		IF stOuterStatus.stOACData.PackCodeStatus[nPackIndex].5 OR stOuterStatus.stOACData.PackCodeStatus[nPackIndex].6 THEN

			FOR nCheckIndex :=1 TO cMAX_PACKS_PER_OUTER DO

				IF stOuterStatus.stOACData.PackCode[nPackIndex] = stLastOuterStatus.stOACData.PackCode[nCheckIndex] THEN

					stOuterStatus.nStatus.22 := TRUE;
					stOuterStatus.sDataSourceTracker  := 'PK_DUPLIC';

					stLastOuterStatus.nStatus.22 := TRUE;
					stLastOuterStatus.sDataSourceTracker  := 'PK_DUPLIC';

					EXIT;
				END_IF
			END_FOR
			EXIT;
		END_IF
	END_FOR
END_IF

bDuplicateFound 	:= FALSE;

(* for dupicats for all packs inside one Outer *)
FOR  nPackIndex :=1 TO cMAX_PACKS_PER_OUTER DO

	IF stOuterStatus.stOACData.PackCodeStatus[nPackIndex].5 OR stOuterStatus.stOACData.PackCodeStatus[nPackIndex].6 THEN

		FOR nCheckIndex := nPackIndex  TO cMAX_PACKS_PER_OUTER DO

			IF stOuterStatus.stOACData.PackCodeStatus[nCheckIndex].5 OR stOuterStatus.stOACData.PackCodeStatus[nCheckIndex].6 THEN

				IF stOuterStatus.stOACData.PackCode[nPackIndex] = stOuterStatus.stOACData.PackCode[nCheckIndex]  AND
					nPackIndex <> nCheckIndex	THEN


					(* duplicate packs found *)
					stOuterStatus.aOACPackStatus[nPackIndex] := 3;
					(*additional bit passing to CAC*)
					stOuterStatus.stOACData.PackCodeStatus[nPackIndex] :=
											F_FiltredSetBitState16(TRUE, 'LOW', 3, TRUE, stOuterStatus.stOACData.PackCodeStatus[nPackIndex]);

					stOuterStatus.aOACPackStatus[nCheckIndex] := 3;
					(*additional bit passing to CAC*)
					stOuterStatus.stOACData.PackCodeStatus[nCheckIndex] :=
											F_FiltredSetBitState16(TRUE, 'LOW', 3, TRUE, stOuterStatus.stOACData.PackCodeStatus[nCheckIndex]);

					bDuplicateFound := TRUE;

					stOuterStatus.stOACData.PackRejectCode[nPackIndex]  	:= stDuplicatedItem.sMetsDisplayCode;
	   				stOuterStatus.stOACData.PackRejectID[nPackIndex] 	 	:= stDuplicatedItem.nRejectID;
					stOuterStatus.stOACData.PackRejectCode[nCheckIndex]  := stDuplicatedItem.sMetsDisplayCode;
					stOuterStatus.stOACData.PackRejectID[nCheckIndex]  	:= stDuplicatedItem.nRejectID;

				END_IF
			END_IF
		END_FOR
	END_IF
END_FOR


IF bDuplicateFound THEN

	nGoodPackReads	:=cMAX_PACKS_PER_OUTER;
	stOuterStatus.nStatus.23 := TRUE;

	FOR  nPackIndex :=1 TO cMAX_PACKS_PER_OUTER DO
		IF stOuterStatus.stOACData.PackCodeStatus[nPackIndex].3 THEN nGoodPackReads := nGoodPackReads - 1; END_IF
	END_FOR

END_IF

END_FUNCTION_BLOCK

// ---- POUs/METS/Common LIB/01_PACK LIB/Pack FBs/FB_PACK_MoveOuterStatusArray.TcPOU
FUNCTION_BLOCK FB_PACK_MoveOuterStatusArray
VAR_INPUT
	bExecute			: BOOL;		(* set TRUE to move array data *)
	bClearShiftReg		: BOOL;		(* set TRUE to clear all array data to 0 *)
END_VAR
VAR_IN_OUT
	aOCVPackStatus			: ARRAY[1..cMAX_OUTER_STATUS_QUEUE] OF ST_OUTER_Status;	(* Outer status register *)
	(*stPackBufferStatusHMI		: ST_HMI_PACK_BufferStatus;*)
END_VAR
VAR_OUTPUT
	bDone						: BOOL;
END_VAR
VAR
	fbExecute			: R_TRIG;
END_VAR

(* rising edge of bShiftReg *)
fbExecute(CLK := bExecute);

(* clear shift reg *)
IF bClearShiftReg = TRUE THEN

	(* reset OCV Outer Status data *)
	MEMSET(ADR(aOCVPackStatus), 16#00, SIZEOF(aOCVPackStatus));

	bDone := FALSE;

(* move shift reg *)
ELSIF fbExecute.Q = TRUE THEN

	(* move OCV Outer Status register [1..cMAX_OUTER_STATUS_QUEUE-1] to [2..cMAX_OUTER_STATUS_QUEUE] *)
	MEMMOVE(ADR(aOCVPackStatus[2]), ADR(aOCVPackStatus[1]), SIZEOF(aOCVPackStatus) - SIZEOF(aOCVPackStatus[1]));
	(* clear OCV Outer Status register [1] *)
	MEMSET(ADR(aOCVPackStatus[1]), 16#00, SIZEOF(aOCVPackStatus[1]));

	(*MEMSET(ADR(stPackBufferStatusHMI), 16#00, SIZEOF(stPackBufferStatusHMI));*)

	bDone := TRUE;

(* no action required, bExecute has been reset *)
ELSIF bExecute = FALSE THEN

	bDone := FALSE;
END_IF

(******************************************************************************************************************************************)
(*
IN CASE OF MULTISHIFT - CAN BE USED THIS:
	nOuterStatusToShift := LIMIT(1, nOuterStatusToShift, cMAX_OUTER_STATUS_QUEUE);
	(* move Outer Status register [1..49] to [2..50] *)
	MEMMOVE(ADR(aOuterStatus[nOuterStatusToShift+1]), ADR(aOuterStatus[1]), SIZEOF(aOuterStatus) - nOuterStatusToShift*SIZEOF(aOuterStatus[1]));
	(* clear Outer Status register [nOuterStatusToShift] *)
	MEMSET(ADR(aOuterStatus[1]), 16#00, nOuterStatusToShift*SIZEOF(aOuterStatus[1]));
*)
(******************************************************************************************************************************************)

END_FUNCTION_BLOCK

// ---- POUs/METS/Common LIB/01_PACK LIB/Pack FBs/FB_PACK_WriteOCVLoopDB.TcPOU
(* scan and validate Outers, generate OAC file for new valid Outers *)
FUNCTION_BLOCK FB_PACK_WriteOCVLoopDB
VAR_INPUT
	bExecute						: BOOL;			(* scan for completed Outer *)
	ePackAggregationMode			: E_SYSTEM_PackAggregationMode ;
	nPacksPerOuter				: INT;
	nPackPos1						: INT 	:=1;
	nPackPos2						: INT	:=2;
	bExtendedDupCheck			: BOOL;
	aDisablePackAggregCamera	: ARRAY[1..3] OF BOOL;
	stDuplicatedItem				: ST_RejectItems;(*stPackRejectReasons.stPackCodesDuplicated*)
	stCTDateTime					: ST_SYSTEM_DateTime;
END_VAR
VAR_IN_OUT
	stOCVDataDB					: ST_DB_OCVDataCtrl;
	stLastOCVDataDB				: ST_DB_OCVDataCtrl;
	stCodeInfo_Pack				: ST_CodeInfo;
	stCodeInfo_Intermediate		: ST_CodeInfo;
	(*aInterimCodeQueue			: ARRAY[1..cMAX_INTERMEDIATE_CODE_QUEUE] OF T_MaxString;*)
	aOCVPackStatus				: ARRAY[1..cMAX_OUTER_STATUS_QUEUE] OF ST_OUTER_Status;	(* Outer status array *)
	stMetsEfficiency				: ST_NOVRAM_METS_Inspection;
	stShiftItemProduced			: ST_KPI_ItemsProduced;
	stProdItemProduced			: ST_KPI_ItemsProduced;
	stLastOCVStatus				: ST_OUTER_Status;	(* Outer status *)
END_VAR
VAR_OUTPUT
	bDone							: BOOL;			(* TRUE = validation complete *)
	bBusy							: BOOL;			(* TRUE = validation in progress *)
	bError							: BOOL;			(* TRUE = validation error *)
	nErrorID						: UDINT;			(* error ID *)

	aOCVRecordDBName			 : ARRAY[1..2] OF T_MaxString;

	bPackCodeDuplicate			: BOOL;
	nLastTriggerID					: UDINT;
	bOCVUpdated					: BOOL;
	bOCVValidated					: BOOL;
	stLastValidatedOCV			: ST_OUTER_Status;	(* Outer status *)
	sPackCodesResultToOCV		: T_LongSTRING;
END_VAR
VAR
	fbExecute					: R_TRIG;
	tonTimeOut				: TON;
	rtTimeOutExec				: R_TRIG;
	eState						: E_OCV_State;
	eErrorState					: E_OCV_State;
	eCodeAIType				: E_CodeAIType;
	nMaxOuterIndex			: INT;
	nOuterIndex				: INT;
	nSourceIndex				: INT;
	nPackIndex				: INT;

	nOCVDataCreated 			: UDINT;
	nOCVStoredInDB 			: UDINT;
	nOCVFaildInDB				: UDINT;
	nLinkedPackInOCV 		: UDINT;

	nOCVUpdatedInDB 		: UDINT;

	bUseIntermediateCode		: BOOL;
	stOCVStatus				: ST_OUTER_Status;	(* Outer status *)

(******************************************************************************)

	fbDuplicatesPackCodesDB		: FB_PACK_DuplicatesPackCodesDB;
	fbPackInspectionEfficency		: FB_KPI_PackEfficiency;

(******************************************************************************)

	aDiagOCVDataDB				: ARRAY[0..1] OF ST_DB_OCVDataCtrl;

	nOCVLogIndex		: T_PositiveINT;
	sAppendedString				: STRING;
	//sLocalTargetPath	: T_MaxString;

END_VAR

(***************************************TimeOut *******************************************)
(* monitor Busy timeout *)
tonTimeOut( IN:=nSourceIndex <> 0, PT:=cONE_SECOND, Q=>);

rtTimeOutExec(CLK:= tonTimeOut.Q);

IF rtTimeOutExec.Q THEN

	bError := TRUE;
	nErrorID := 100;
	IF nSourceIndex > 0 THEN

		aOCVPackStatus[nSourceIndex].sDataSourceTracker 	:= 	'TIMEOUT_S';
		aOCVPackStatus[nSourceIndex].nStatus.7 := TRUE;

		stLastOCVStatus := aOCVPackStatus[nSourceIndex];
		bOCVUpdated	:= TRUE;
		sPackCodesResultToOCV	:= 'TIMEOUT_OCV';

		stLastValidatedOCV := aOCVPackStatus[nSourceIndex];
		bOCVValidated	:= TRUE;
	END_IF

	MEMSET(ADR(stOCVDataDB), 16#00, SIZEOF(stOCVDataDB));
	MEMSET(ADR(stLastOCVDataDB), 16#00, SIZEOF(stLastOCVDataDB));


	eState := E_OCV_DONE;
END_IF

(***************************************Execution*******************************************)

(* monitor rising edge of bExecute *)
fbExecute(CLK := bExecute);

(* rising edge of bExecute *)
CASE eState OF

	(* idle *)
	E_OCV_IDLE:

		(* scan for completed Outer when OAC files are required *)
		IF fbExecute.Q = TRUE THEN

			(* update outputs *)
			bDone := FALSE;
			bBusy := TRUE;
			bError := FALSE;
			nErrorID := 0;

			(* clear outputs *)
			nOCVDataCreated 		:= 0;
			nOCVStoredInDB 		:= 0;
			nOCVFaildInDB			:= 0;
			nLinkedPackInOCV 	:= 0;


			(*bOCVUpdated	:= FALSE;*)

			(* max Outer index *)
			nMaxOuterIndex := UDINT_TO_INT(SIZEOF(aOCVPackStatus) / SIZEOF(aOCVPackStatus[1]));

			eState := E_OCV_SCAN;

		(* no action required *)
		ELSIF bExecute = FALSE THEN

			(* reset outputs *)
			bDone := FALSE;
			bBusy := FALSE;
			bError := FALSE;
			nErrorID := 0;

		END_IF

	(* scan for completed Outer *)
	E_OCV_SCAN:

		eState := E_OCV_DONE;
		bOCVUpdated	:= FALSE;
		bOCVValidated	:= FALSE;

		(* reset index of Outer to be written to OCV file *)
		nSourceIndex := 0;

		aOCVRecordDBName[1] := '';
		aOCVRecordDBName[2] := '';

		bPackCodeDuplicate			:= FALSE;

		 (* scan aOCVPackStatus  backward - ensures that oldest Outer will be written first *)
		FOR nOuterIndex := nMaxOuterIndex TO 1 BY -1 DO
			CASE ePackAggregationMode OF

			E_SYSTEM_PAOL_3CAM:
				(* TriggerID > 0 indicates Outer data present, nStatus = 14 indicates writing data for all 3 cameras, nStatus.6  indicates OCV file has been alread  created, nStatus.7 indicates OCV write error  *)
				IF aOCVPackStatus[nOuterIndex].nTriggerID > 0 AND
					(aOCVPackStatus[nOuterIndex].nStatus.1 OR aDisablePackAggregCamera[1])	AND
					( aOCVPackStatus[nOuterIndex].nStatus.2 OR aDisablePackAggregCamera[2]) 	AND
					( aOCVPackStatus[nOuterIndex].nStatus.3 OR aDisablePackAggregCamera[3]) 	AND
					NOT aOCVPackStatus[nOuterIndex].nStatus.6 		AND
					NOT aOCVPackStatus[nOuterIndex].nStatus.7  		(*AND
					NOT aOCVPackStatus[nOuterIndex].nStatus.22		AND
					NOT aOCVPackStatus[nOuterIndex].nStatus.23 *)	THEN

					(* For lightbox system,mapping packcodes to AggregationCodes, used for file name has to be done here, when we are sure if all pack data was plced to OCV record. Those codes will be used to restore OCV data to OAC*)
					AggregationCodes();

					bUseIntermediateCode := FALSE;
					nSourceIndex := nOuterIndex;
					EXIT;
				END_IF

			E_SYSTEM_PAOL_2CAM:
				(* TriggerID > 0 indicates Outer data present, nStatus = 14 indicates writing data for all 3 cameras, nStatus.6  indicates OCV file has been alread  created, nStatus.7 indicates OCV write error  *)
				IF aOCVPackStatus[nOuterIndex].nTriggerID > 0 AND
					(aOCVPackStatus[nOuterIndex].nStatus.1 OR aDisablePackAggregCamera[1])		AND
					( aOCVPackStatus[nOuterIndex].nStatus.2 OR aDisablePackAggregCamera[2]) 	AND
					NOT aOCVPackStatus[nOuterIndex].nStatus.6 		AND
					NOT aOCVPackStatus[nOuterIndex].nStatus.7  		(*AND
					NOT aOCVPackStatus[nOuterIndex].nStatus.22		AND
					NOT aOCVPackStatus[nOuterIndex].nStatus.23*) 	THEN

					(* For lightbox system,mapping packcodes to AggregationCodes, used for file name has to be done here, when we are sure if all pack data was plced to OCV record. Those codes will be used to restore OCV data to OAC*)
					AggregationCodes();

					bUseIntermediateCode := FALSE;
					nSourceIndex := nOuterIndex;
					EXIT;
				END_IF

			E_SYSTEM_PLAS_T01:
				(* TriggerID > 0 indicates Outer data present, nStatus = 14 indicates writing data for all 3 cameras, nStatus.6  indicates OCV file has been alread  created, nStatus.7 indicates OCV write error  *)
				(* For linear aggregation system,AggregationCode shuld be already add from temporary coding system camera. This code will be used for file name and to restore OCV data to OAC*)

				IF aOCVPackStatus[nOuterIndex].nTriggerID > 0 		AND
					aOCVPackStatus[nOuterIndex].nStatus.0			AND 	(*OCV Structure rady to store in file *)
					NOT aOCVPackStatus[nOuterIndex].nStatus.6 		AND
					NOT aOCVPackStatus[nOuterIndex].nStatus.7  		(*AND
					NOT aOCVPackStatus[nOuterIndex].nStatus.22		AND
					NOT aOCVPackStatus[nOuterIndex].nStatus.23 *)	THEN

					(* For clear wrap system,mapping packcodes to AggregationCodes, used for file name has to be done here, when we are sure if all pack data was plced to OCV record. Those codes will be used to restore OCV data to OAC*)
					AggregationCodes();

					bUseIntermediateCode := FALSE;
					nSourceIndex := nOuterIndex;
					EXIT;
				END_IF

			E_SYSTEM_PLAS_T02, E_SYSTEM_PLAS_T03, E_SYSTEM_PLAS_T04:
				(* TriggerID > 0 indicates Outer data present, nStatus = 14 indicates writing data for all 3 cameras, nStatus.6  indicates OCV file has been alread  created, nStatus.7 indicates OCV write error  *)
				(* For linear aggregation system,AggregationCode shuld be already add from temporary coding system camera. This code will be used for file name and to restore OCV data to OAC*)

				IF aOCVPackStatus[nOuterIndex].nTriggerID > 0 		AND
					aOCVPackStatus[nOuterIndex].nStatus.0			AND 	(*OCV Structure rady to store in file *)
					NOT aOCVPackStatus[nOuterIndex].nStatus.6 		AND
					NOT aOCVPackStatus[nOuterIndex].nStatus.7  		(*AND
					NOT aOCVPackStatus[nOuterIndex].nStatus.22		AND
					NOT aOCVPackStatus[nOuterIndex].nStatus.23 *)	THEN

					(* For NON clear wrap system,mapping packcodes to AggregationCodes form Intrim code, which might be temp stored as barcode for OCV records.
						AggregationCode1 will be used for file name has to be done here, when we are sure if all pack data was plced to OCV record. Those codes will be used to restore OCV data to OAC*)
						(*aOCVPackStatus[nOuterIndex].stOACData.AggregationCodes[1] :=aOCVPackStatus[nOuterIndex].stOACData.Barcode;*) (*solution never tested yet*)

					bUseIntermediateCode := TRUE;
					nSourceIndex := nOuterIndex;
					EXIT;
				END_IF
			END_CASE
		END_FOR

		(* Outer found requiring OAC file to be written *)
		IF nSourceIndex > 0 THEN

			(* copy Outer data from arrOuterStatus *)
			stOCVStatus := aOCVPackStatus[nSourceIndex];

			fbDuplicatesPackCodesDB(
				stDuplicatedItem := stDuplicatedItem,
				bExtendedDupCheck	:=	bExtendedDupCheck,
				stOuterStatus := stOCVStatus,
				stLastOuterStatus := aOCVPackStatus[nSourceIndex+1],
				bDuplicateFound =>  bPackCodeDuplicate
				);

			stMetsEfficiency.OutersProcessing.AtPackAggregCameras := stMetsEfficiency.OutersProcessing.AtPackAggregCameras  + 1;

			fbPackInspectionEfficency(
				ePackAggregationMode				:= ePackAggregationMode,
				nTotalOutersProcessingByPackAggregCameras	:= stMetsEfficiency.OutersProcessing.AtPackAggregCameras,
				bUseInterimCode						:= bUseIntermediateCode,
				sOuterStatus							:= stOCVStatus,
				aPacksRead							:= stMetsEfficiency.PacksRead,
				aPackPosEfficiency						:= stMetsEfficiency.PackPosEfficiency,
				stPackAggregationEfficiency			:= stMetsEfficiency.PackAggregationEfficiency,
				stMainItemProduced					:= stMetsEfficiency.PackProduced,
				stShiftItemProduced					:= stShiftItemProduced,
				stProdItemProduced					:= stProdItemProduced
				);

			nOCVDataCreated := nOCVDataCreated +1;

			stLastValidatedOCV := stOCVStatus; (*Use for logging data*)
			bOCVValidated	:= TRUE;	(*Use for SFLX solution*)

			IF aOCVPackStatus[nSourceIndex+1].nStatus.22 AND stOCVStatus.nStatus.22  AND nSourceIndex <  nMaxOuterIndex  THEN

				stLastOCVDataDB.stOCVStatusDB	:= aOCVPackStatus[nSourceIndex+1];
				stLastOCVDataDB.bBlockRecord	:= TRUE;
				stLastOCVDataDB.bUpdateDataReq 	:= TRUE;

				eState := E_OCV_UPDATEDATA;
			ELSE
				eState := E_OCV_WRITEDATA;
			END_IF
		END_IF

	E_OCV_UPDATEDATA:

		IF	stLastOCVDataDB.bDone	THEN

			IF NOT  stLastOCVDataDB.bError THEN

				nOCVUpdatedInDB := nOCVUpdatedInDB +1;
			ELSE
				bError := TRUE;
				nErrorID := stLastOCVDataDB.nErrorID;
				eErrorState := eState;
			END_IF

			aDiagOCVDataDB[1]	:= stLastOCVDataDB;

			eState := E_OCV_WRITEDATA;
		END_IF

	E_OCV_WRITEDATA:

		IF F_InvalidateASCIIChar(F_CODE_GetItem(stOCVStatus.stOACData.AggregationCodes[1] , eCodeAIType.SerialCode, SEL(bUseIntermediateCode, stCodeInfo_Pack, stCodeInfo_Intermediate))) >	0 	THEN

			stOCVStatus.sDataSourceTracker  := 'AGG_INVAL';
			stOCVStatus.nStatus.22 := TRUE;
		ELSE
			stOCVDataDB.sFileCodeName1	:= F_CodeToHex(F_CODE_GetItem(stOCVStatus.stOACData.AggregationCodes[1] , eCodeAIType.SerialCode, SEL(bUseIntermediateCode, stCodeInfo_Pack, stCodeInfo_Intermediate)));
		END_IF

		IF F_InvalidateASCIIChar(F_CODE_GetItem(stOCVStatus.stOACData.AggregationCodes[2] , eCodeAIType.SerialCode,   stCodeInfo_Pack)) >	0 	THEN

			stOCVStatus.sDataSourceTracker  := 'AGG_INVAL';
			stOCVStatus.nStatus.22 := TRUE;
		ELSE
			stOCVDataDB.sFileCodeName2	:= F_CodeToHex(F_CODE_GetItem(stOCVStatus.stOACData.AggregationCodes[2] , eCodeAIType.SerialCode,   stCodeInfo_Pack)); (*no reason to have 2 diffrent intermediate codes*)
		END_IF

		IF stOCVStatus.nStatus.22 THEN
			stOCVDataDB.bBlockRecord	:= TRUE;
		END_IF
		stOCVDataDB.stOCVStatusDB	:= stOCVStatus;
		stOCVDataDB.bCreateDataReq 	:= TRUE;

(*Place for HectorDB block*)

		IF	stOCVDataDB.bDone	THEN

			aOCVRecordDBName[1] := stOCVDataDB.sFileCodeName1;
			aOCVRecordDBName[2] := stOCVDataDB.sFileCodeName2;

			IF NOT  stOCVDataDB.bError THEN
				nLastTriggerID :=  stOCVStatus.nTriggerID;
				nOCVStoredInDB := nOCVStoredInDB +1;
				(* update stOCVStatus - OCV file written OK *)
				stOCVStatus.nStatus.6 := TRUE;

			ELSE
				bError := TRUE;
				nErrorID := stOCVDataDB.nErrorID;
				nOCVFaildInDB := nOCVFaildInDB +1;
				(* update stOCVStatus - OCV file write error  - general error for OCV *)
				stOCVStatus.nStatus.7 := TRUE;
				eErrorState := eState;
			END_IF

			aDiagOCVDataDB[0]	:= stOCVDataDB;

			eState := E_OCV_UPDATESTATUS;
		END_IF

	(* update Outer status *)
	E_OCV_UPDATESTATUS:

		MEMSET(ADR(stOCVDataDB), 16#00, SIZEOF(stOCVDataDB));
		MEMSET(ADR(stLastOCVDataDB), 16#00, SIZEOF(stLastOCVDataDB));

		nSourceIndex := 0;
		(* move stOCVStatus data back to shift reg *)
		FOR nOuterIndex := 1 TO nMaxOuterIndex DO

			(* matching nTriggerID found *)
			IF aOCVPackStatus[nOuterIndex].nTriggerID = stOCVStatus.nTriggerID THEN

				(* move updated Outer data to shift reg *)
				aOCVPackStatus[nOuterIndex] := stOCVStatus;
				stLastOCVStatus := stOCVStatus;

				nLinkedPackInOCV :=nLinkedPackInOCV + TO_UDINT(stOCVStatus.stOACData.NumberOfLinkedPacks);
				bOCVUpdated	:= TRUE;
				
				sAppendedString			:= '';
				sPackCodesResultToOCV	:= '';
				
				sPackCodesResultToOCV := F_CONCAT5('[', RIGHT(stLastOCVStatus.stOACData.AggregationCodes[1],7),']:[',RIGHT(stLastOCVStatus.stOACData.AggregationCodes[2],7),']');
				FOR nOCVLogIndex := 1 TO MIN(nPacksPerOuter ,cMAX_PACKS_PER_OUTER) BY 1 DO
					//sPackCodesResultToOCV :=F_LongCONCAT(sPackCodesResultToOCV, '     ');
					//sPackCodesResultToOCV := F_LongCONCAT(sPackCodesResultToOCV, RIGHT(F_CODE_GetItem(stLastOCVStatus.stOACData.PackCode[nOCVLogIndex], eCodeAIType.SerialCode, stCodeInfo_Pack),7));
					
					CONCAT2(ADR(sPackCodesResultToOCV), ADR('   '), ADR(sPackCodesResultToOCV), SIZEOF(sPackCodesResultToOCV));
		
					sAppendedString := RIGHT(F_CODE_GetItem(stLastOCVStatus.stOACData.PackCode[nOCVLogIndex], eCodeAIType.SerialCode, stCodeInfo_Pack),7);
					CONCAT2(ADR(sPackCodesResultToOCV), ADR(sAppendedString), ADR(sPackCodesResultToOCV), SIZEOF(sPackCodesResultToOCV));

				END_FOR

				EXIT;
			END_IF
		END_FOR

		eState := E_OCV_SCAN;

	(* OCV file complete *)
	E_OCV_DONE:

		(* update outputs *)
		bDone := TRUE;
		bBusy := FALSE;

		eState := E_OCV_IDLE;

(* unknown state *)
ELSE

	eState := E_OCV_IDLE;
END_CASE

ACTION AggregationCodes:
IF nPackPos1 > 0 AND  nPackPos1 <= cMAX_PACKS_PER_OUTER THEN
	IF NOT aOCVPackStatus[nOuterIndex].stOACData.PackCodeStatus[nPackPos1].0 AND
		NOT aOCVPackStatus[nOuterIndex].stOACData.PackCodeStatus[nPackPos1].1 THEN

		aOCVPackStatus[nOuterIndex].stOACData.AggregationCodes[1] :=aOCVPackStatus[nOuterIndex].stOACData.PackCode[nPackPos1];
	ELSE
		aOCVPackStatus[nOuterIndex].stOACData.AggregationCodes[1] := '';
	END_IF
ELSE
	aOCVPackStatus[nOuterIndex].stOACData.AggregationCodes[1] := '';
END_IF

IF nPackPos2 > 0 AND  nPackPos2 <= cMAX_PACKS_PER_OUTER  THEN
	IF NOT aOCVPackStatus[nOuterIndex].stOACData.PackCodeStatus[nPackPos2].0 AND
		NOT aOCVPackStatus[nOuterIndex].stOACData.PackCodeStatus[nPackPos2].1 THEN

		aOCVPackStatus[nOuterIndex].stOACData.AggregationCodes[2] :=aOCVPackStatus[nOuterIndex].stOACData.PackCode[nPackPos2];
	ELSE
		aOCVPackStatus[nOuterIndex].stOACData.AggregationCodes[2] := '';
	END_IF
ELSE
	aOCVPackStatus[nOuterIndex].stOACData.AggregationCodes[2] := '';
END_IF
END_ACTION

END_FUNCTION_BLOCK

// ---- POUs/METS/Common LIB/06_KPI LIB/ItemEfficiency/FB_KPI_PackEfficiency.TcPOU
FUNCTION_BLOCK FB_KPI_PackEfficiency
VAR_INPUT
	ePackAggregationMode							: E_SYSTEM_PackAggregationMode ;
	nTotalOutersProcessingByPackAggregCameras	: UDINT;
	bUseInterimCode									: BOOL;
END_VAR
VAR_IN_OUT
	sOuterStatus							: ST_OUTER_Status;	(* Outer status *)
	aPacksRead							: ARRAY[0..cMAX_PACKS_PER_OUTER] OF UDINT;
	aPackPosEfficiency						: ARRAY[1..cMAX_PACKS_PER_OUTER] OF ST_KPI_CodePos;
	stPackAggregationEfficiency				: ST_KPI_InspectionEfficency;
	stMainItemProduced					: ST_KPI_ItemsProduced;
	stShiftItemProduced						: ST_KPI_ItemsProduced;
	stProdItemProduced					: ST_KPI_ItemsProduced;
END_VAR
VAR
	nPackPositionIndex						: INT;
	bValidOuter							: BOOL;
	nTestCountPLAS			: INT;
	nTestCountPAOL			: INT;
	nTestCount2CAM			: INT;
END_VAR

CASE ePackAggregationMode OF

	E_SYSTEM_PAOL_2CAM:

		CAM2();

	E_SYSTEM_PAOL_3CAM:

		PAOL();

	E_SYSTEM_PLAS_T01, E_SYSTEM_PLAS_T02, E_SYSTEM_PLAS_T03, E_SYSTEM_PLAS_T04:

		PLAS();

END_CASE

ACTION CAM2:
nTestCount2CAM := nTestCount2CAM + 1;

bValidOuter := TRUE;

IF sOuterStatus.stOACData.NumberOfLinkedPacks <= cMAX_PACKS_PER_OUTER AND
	sOuterStatus.stOACData.NumberOfLinkedPacks >=0 THEN

	aPacksRead[sOuterStatus.stOACData.NumberOfLinkedPacks] := aPacksRead[sOuterStatus.stOACData.NumberOfLinkedPacks] +1;
END_IF

IF sOuterStatus.stOACData.NumberOfPacks <= cMAX_PACKS_PER_OUTER AND
	sOuterStatus.stOACData.NumberOfPacks >=0 THEN

	FOR nPackPositionIndex := 1 TO sOuterStatus.stOACData.NumberOfPacks DO
		(* Pack code is valid *)
		IF sOuterStatus.aOACPackStatus[nPackPositionIndex] = 5  THEN
	
			aPackPosEfficiency[nPackPositionIndex].ReadOK := aPackPosEfficiency[nPackPositionIndex].ReadOK + 1;
	
			stMainItemProduced.Passed:= stMainItemProduced.Passed + 1;
			stShiftItemProduced.Passed:= stShiftItemProduced.Passed + 1;
			stProdItemProduced.Passed:= stProdItemProduced.Passed + 1;
		ELSE
	
			bValidOuter := FALSE;
	
			stMainItemProduced.Rejected := stMainItemProduced.Rejected + 1;
			stShiftItemProduced.Rejected := stShiftItemProduced.Rejected + 1;
			stProdItemProduced.Rejected := stProdItemProduced.Rejected + 1;
		END_IF
	
		stMainItemProduced.Total := stMainItemProduced.Total+ 1;
		stShiftItemProduced.Total := stShiftItemProduced.Total+ 1;
		stProdItemProduced.Total := stProdItemProduced.Total+ 1;
	
		(* update read efficiency for indyvidual Pack position *)
		aPackPosEfficiency[nPackPositionIndex].Efficiency := F_SafeDIV(UDINT_TO_LREAL(aPackPosEfficiency[nPackPositionIndex].ReadOK),
																			UDINT_TO_LREAL(nTotalOutersProcessingByPackAggregCameras )) * 100.0;
		aPackPosEfficiency[nPackPositionIndex].Efficiency  :=LIMIT(0, aPackPosEfficiency[nPackPositionIndex].Efficiency , 100);
	END_FOR
END_IF

stPackAggregationEfficiency.ProcessedTotal := stPackAggregationEfficiency.ProcessedTotal + 1;

IF bValidOuter THEN
	stPackAggregationEfficiency.ProcessedSuccessful := stPackAggregationEfficiency.ProcessedSuccessful + 1;
ELSE
	stPackAggregationEfficiency.ProcessedRejected := stPackAggregationEfficiency.ProcessedRejected + 1;
END_IF

stPackAggregationEfficiency.ProcessedEfficiency := F_SafeDIV(UDINT_TO_LREAL(stPackAggregationEfficiency.ProcessedSuccessful),
																	UDINT_TO_LREAL(stPackAggregationEfficiency.ProcessedTotal )) * 100.0;
stPackAggregationEfficiency.ProcessedEfficiency  :=LIMIT(0, stPackAggregationEfficiency.ProcessedEfficiency , 100);

stMainItemProduced.Efficiency := F_SafeDIV(stMainItemProduced.Passed * 100, stMainItemProduced.Total);
stMainItemProduced.Efficiency :=LIMIT(0, stMainItemProduced.Efficiency, 100);

stShiftItemProduced.Efficiency := F_SafeDIV(stShiftItemProduced.Passed * 100, stShiftItemProduced.Total);
stShiftItemProduced.Efficiency :=LIMIT(0, stShiftItemProduced.Efficiency, 100);

stProdItemProduced.Efficiency := F_SafeDIV(stProdItemProduced.Passed * 100, stProdItemProduced.Total);
stProdItemProduced.Efficiency :=LIMIT(0, stProdItemProduced.Efficiency, 100);
END_ACTION

ACTION NCW:
aPacksRead[sOuterStatus.stOACData.NumberOfLinkedPacks] := aPacksRead[sOuterStatus.stOACData.NumberOfLinkedPacks] +1;

FOR nPackPositionIndex := 1 TO sOuterStatus.stOACData.NumberOfPacks DO
	(* Pack code is valid *)
	IF sOuterStatus.aOACPackStatus[nPackPositionIndex] = 5 THEN

		aPackPosEfficiency[nPackPositionIndex].ReadOK := aPackPosEfficiency[nPackPositionIndex].ReadOK + 1;

		stMainItemProduced.Passed:= stMainItemProduced.Passed + 1;
		stShiftItemProduced.Passed:= stShiftItemProduced.Passed + 1;
		stProdItemProduced.Passed:= stProdItemProduced.Passed + 1;
	ELSE

		stMainItemProduced.Rejected := stMainItemProduced.Rejected + 1;
		stShiftItemProduced.Rejected := stShiftItemProduced.Rejected + 1;
		stProdItemProduced.Rejected := stProdItemProduced.Rejected + 1;
	END_IF

	stMainItemProduced.Total := stMainItemProduced.Total+ 1;
	stShiftItemProduced.Total := stShiftItemProduced.Total+ 1;
	stProdItemProduced.Total := stProdItemProduced.Total+ 1;

	(* update read efficiency for indyvidual Pack position *)
	aPackPosEfficiency[nPackPositionIndex].Efficiency := F_SafeDIV(UDINT_TO_LREAL(aPackPosEfficiency[nPackPositionIndex].ReadOK),
																		UDINT_TO_LREAL(nTotalOutersProcessingByPackAggregCameras )) * 100.0;
	aPackPosEfficiency[nPackPositionIndex].Efficiency  :=LIMIT(0, aPackPosEfficiency[nPackPositionIndex].Efficiency , 100);
END_FOR

stMainItemProduced.Efficiency := F_SafeDIV(stMainItemProduced.Passed * 100, stMainItemProduced.Total);
stMainItemProduced.Efficiency :=LIMIT(0, stMainItemProduced.Efficiency, 100);

stShiftItemProduced.Efficiency := F_SafeDIV(stShiftItemProduced.Passed * 100, stShiftItemProduced.Total);
stShiftItemProduced.Efficiency :=LIMIT(0, stShiftItemProduced.Efficiency, 100);

stProdItemProduced.Efficiency := F_SafeDIV(stProdItemProduced.Passed * 100, stProdItemProduced.Total);
stProdItemProduced.Efficiency :=LIMIT(0, stProdItemProduced.Efficiency, 100);
END_ACTION

ACTION PAOL:
nTestCountPAOL := nTestCountPAOL + 1;

bValidOuter := TRUE;

IF sOuterStatus.stOACData.NumberOfLinkedPacks <= cMAX_PACKS_PER_OUTER AND
	sOuterStatus.stOACData.NumberOfLinkedPacks >=0 THEN

	aPacksRead[sOuterStatus.stOACData.NumberOfLinkedPacks] := aPacksRead[sOuterStatus.stOACData.NumberOfLinkedPacks] +1;
END_IF

IF sOuterStatus.stOACData.NumberOfPacks <= cMAX_PACKS_PER_OUTER AND
	sOuterStatus.stOACData.NumberOfPacks >=0 THEN

	FOR nPackPositionIndex := 1 TO sOuterStatus.stOACData.NumberOfPacks DO
		(* Pack code is valid *)
		IF sOuterStatus.aOACPackStatus[nPackPositionIndex] = 5  THEN
	
			aPackPosEfficiency[nPackPositionIndex].ReadOK := aPackPosEfficiency[nPackPositionIndex].ReadOK + 1;
	
			stMainItemProduced.Passed:= stMainItemProduced.Passed + 1;
			stShiftItemProduced.Passed:= stShiftItemProduced.Passed + 1;
			stProdItemProduced.Passed:= stProdItemProduced.Passed + 1;
		ELSE
	
			bValidOuter := FALSE;
	
			stMainItemProduced.Rejected := stMainItemProduced.Rejected + 1;
			stShiftItemProduced.Rejected := stShiftItemProduced.Rejected + 1;
			stProdItemProduced.Rejected := stProdItemProduced.Rejected + 1;
		END_IF
	
		stMainItemProduced.Total := stMainItemProduced.Total+ 1;
		stShiftItemProduced.Total := stShiftItemProduced.Total+ 1;
		stProdItemProduced.Total := stProdItemProduced.Total+ 1;
	
		(* update read efficiency for indyvidual Pack position *)
		aPackPosEfficiency[nPackPositionIndex].Efficiency := F_SafeDIV(UDINT_TO_LREAL(aPackPosEfficiency[nPackPositionIndex].ReadOK),
																			UDINT_TO_LREAL(nTotalOutersProcessingByPackAggregCameras )) * 100.0;
		aPackPosEfficiency[nPackPositionIndex].Efficiency  :=LIMIT(0, aPackPosEfficiency[nPackPositionIndex].Efficiency , 100);
	END_FOR
END_IF

stPackAggregationEfficiency.ProcessedTotal := stPackAggregationEfficiency.ProcessedTotal + 1;

IF bValidOuter THEN
	stPackAggregationEfficiency.ProcessedSuccessful := stPackAggregationEfficiency.ProcessedSuccessful + 1;
ELSE
	stPackAggregationEfficiency.ProcessedRejected := stPackAggregationEfficiency.ProcessedRejected + 1;
END_IF

stPackAggregationEfficiency.ProcessedEfficiency := F_SafeDIV(UDINT_TO_LREAL(stPackAggregationEfficiency.ProcessedSuccessful),
																	UDINT_TO_LREAL(stPackAggregationEfficiency.ProcessedTotal )) * 100.0;
stPackAggregationEfficiency.ProcessedEfficiency  :=LIMIT(0, stPackAggregationEfficiency.ProcessedEfficiency , 100);

stMainItemProduced.Efficiency := F_SafeDIV(stMainItemProduced.Passed * 100, stMainItemProduced.Total);
stMainItemProduced.Efficiency :=LIMIT(0, stMainItemProduced.Efficiency, 100);

stShiftItemProduced.Efficiency := F_SafeDIV(stShiftItemProduced.Passed * 100, stShiftItemProduced.Total);
stShiftItemProduced.Efficiency :=LIMIT(0, stShiftItemProduced.Efficiency, 100);

stProdItemProduced.Efficiency := F_SafeDIV(stProdItemProduced.Passed * 100, stProdItemProduced.Total);
stProdItemProduced.Efficiency :=LIMIT(0, stProdItemProduced.Efficiency, 100);
END_ACTION

ACTION PLAS:
nTestCountPLAS := nTestCountPLAS + 1;

bValidOuter := TRUE;

IF sOuterStatus.stOACData.NumberOfPacks <= cMAX_PACKS_PER_OUTER AND
	sOuterStatus.stOACData.NumberOfPacks >=0 THEN

	FOR nPackPositionIndex := 1 TO sOuterStatus.stOACData.NumberOfPacks DO
	
		(* Pack code restored from masterlist, by position *)
		IF sOuterStatus.aOACPackStatus[nPackPositionIndex] = 6  THEN
			aPacksRead[nPackPositionIndex] := aPacksRead[nPackPositionIndex] +1;
		END_IF

		(* Pack code is valid *)
		IF sOuterStatus.aOACPackStatus[nPackPositionIndex] = 5
			OR  sOuterStatus.aOACPackStatus[nPackPositionIndex] = 6  THEN
	
			aPackPosEfficiency[nPackPositionIndex].ReadOK := aPackPosEfficiency[nPackPositionIndex].ReadOK + 1;
	
			stMainItemProduced.Passed:= stMainItemProduced.Passed + 1;
			stShiftItemProduced.Passed:= stShiftItemProduced.Passed + 1;
			stProdItemProduced.Passed:= stProdItemProduced.Passed + 1;
		ELSE

			bValidOuter := FALSE;
	
			stMainItemProduced.Rejected := stMainItemProduced.Rejected + 1;
			stShiftItemProduced.Rejected := stShiftItemProduced.Rejected + 1;
			stProdItemProduced.Rejected := stProdItemProduced.Rejected + 1;
		END_IF
	
		stMainItemProduced.Total := stMainItemProduced.Total+ 1;
		stShiftItemProduced.Total := stShiftItemProduced.Total+ 1;
		stProdItemProduced.Total := stProdItemProduced.Total+ 1;
	
		(* update read efficiency for indyvidual Pack position *)
		aPackPosEfficiency[nPackPositionIndex].Efficiency := F_SafeDIV(UDINT_TO_LREAL(aPackPosEfficiency[nPackPositionIndex].ReadOK),
																			UDINT_TO_LREAL(nTotalOutersProcessingByPackAggregCameras )) * 100.0;
		aPackPosEfficiency[nPackPositionIndex].Efficiency  :=LIMIT(0, aPackPosEfficiency[nPackPositionIndex].Efficiency , 100);
	END_FOR
END_IF
(******************************************************************************************************************************************)

stPackAggregationEfficiency.ProcessedTotal := stPackAggregationEfficiency.ProcessedTotal + 1;

IF (sOuterStatus.stOACData.AggregationCodes[1] = cCODE_OVERWIRTTEN OR
		sOuterStatus.stOACData.AggregationCodes[1] = '')		AND
		bUseInterimCode 											THEN

	bValidOuter := FALSE;
END_IF

IF bValidOuter THEN
	stPackAggregationEfficiency.ProcessedSuccessful := stPackAggregationEfficiency.ProcessedSuccessful + 1;
ELSE
	stPackAggregationEfficiency.ProcessedRejected := stPackAggregationEfficiency.ProcessedRejected + 1;
END_IF

stPackAggregationEfficiency.ProcessedEfficiency := F_SafeDIV(UDINT_TO_LREAL(stPackAggregationEfficiency.ProcessedSuccessful),
																	UDINT_TO_LREAL(stPackAggregationEfficiency.ProcessedTotal )) * 100.0;
stPackAggregationEfficiency.ProcessedEfficiency  :=LIMIT(0, stPackAggregationEfficiency.ProcessedEfficiency , 100);

(******************************************************************************************************************************************)

stMainItemProduced.Efficiency := F_SafeDIV(stMainItemProduced.Passed * 100, stMainItemProduced.Total);
stMainItemProduced.Efficiency :=LIMIT(0, stMainItemProduced.Efficiency, 100);

stShiftItemProduced.Efficiency := F_SafeDIV(stShiftItemProduced.Passed * 100, stShiftItemProduced.Total);
stShiftItemProduced.Efficiency :=LIMIT(0, stShiftItemProduced.Efficiency, 100);

stProdItemProduced.Efficiency := F_SafeDIV(stProdItemProduced.Passed * 100, stProdItemProduced.Total);
stProdItemProduced.Efficiency :=LIMIT(0, stProdItemProduced.Efficiency, 100);
END_ACTION

END_FUNCTION_BLOCK

// ---- POUs/METS/Common LIB/08_SOFTWARE LIB/Maths FBs/F_SafeDIV.TcPOU
(* F_SafeDiv prevents PLC crash with DIV0 error by pre-checking that the denominator <> 0 *)
(* Value of 0 is returned if denominator = 0 *)
FUNCTION F_SafeDIV : LREAL
VAR_INPUT
	fNumerator		: LREAL;
	fDenominator	: LREAL;
END_VAR
(*
-------------------------------------------------------------------------------------------------
Date		Version	Author	Comments
-------------------------------------------------------------------------------------------------
30/01/2015	3.00.00	PB		LREAL now used in place of REAL

-------------------------------------------------------------------------------------------------
05/02/10	1.00.00	PB		Initial release

-------------------------------------------------------------------------------------------------
*)

(* do not perform DIV if Denominator = 0 *)
IF fDenominator = 0 THEN

	F_SafeDIV := 0;

(* safe to perform DIV *)
ELSE

	F_SafeDIV := fNumerator / fDenominator;
END_IF

END_FUNCTION

// ---- POUs/METS/Common LIB/01_PACK LIB/Pack Functions/F_PACK_GetRejectReasonFSS.TcPOU
FUNCTION F_PACK_GetRejectReasonFSS : T_FSS_RejecCode
VAR_INPUT
	sRejectReasonME			:	STRING(255);
	stPackRejectReasons		: ST_RejectReasonsForPack;
END_VAR
VAR
	sRejectReasonFSS	: T_FSS_RejecCode;
END_VAR

IF sRejectReasonME = 'OK' THEN
	sRejectReasonFSS := '';

ELSIF sRejectReasonME = '' THEN
	sRejectReasonFSS := stPackRejectReasons.stPackCodesNotLinked.sFssSendCode;

ELSIF FIND(sRejectReasonME, stPackRejectReasons.stPackCodesOverwritten.sMetsSearchCode) > 0 THEN
	sRejectReasonFSS := stPackRejectReasons.stPackCodesOverwritten.sFssSendCode;

ELSIF FIND(sRejectReasonME, stPackRejectReasons.stPackCodesGtinError.sMetsSearchCode) > 0 THEN
	sRejectReasonFSS := stPackRejectReasons.stPackCodesGtinError.sFssSendCode;

ELSIF FIND(sRejectReasonME, stPackRejectReasons.stPackCodesSerialError.sMetsSearchCode) > 0 THEN
	sRejectReasonFSS := stPackRejectReasons.stPackCodesSerialError.sFssSendCode;

ELSIF FIND(sRejectReasonME, stPackRejectReasons.stPackCodeInvalidLength.sMetsSearchCode) > 0 THEN
	sRejectReasonFSS := stPackRejectReasons.stPackCodeInvalidLength.sFssSendCode;

ELSIF FIND(sRejectReasonME, stPackRejectReasons.stPackCodesNotRead.sMetsSearchCode) > 0 THEN
	sRejectReasonFSS := stPackRejectReasons.stPackCodesNotRead.sFssSendCode;

ELSIF FIND(sRejectReasonME, stPackRejectReasons.stPackCodesDuplicated.sMetsSearchCode) > 0 THEN
	sRejectReasonFSS := stPackRejectReasons.stPackCodesDuplicated.sFssSendCode;

ELSIF FIND(sRejectReasonME, stPackRejectReasons.stPackCodesTypeError.sMetsSearchCode) > 0 THEN
	sRejectReasonFSS := stPackRejectReasons.stPackCodesTypeError.sFssSendCode;

ELSIF FIND(sRejectReasonME, stPackRejectReasons.stPackCodesSUPIError.sMetsSearchCode) > 0 THEN
	sRejectReasonFSS := stPackRejectReasons.stPackCodesSUPIError.sFssSendCode;

ELSIF FIND(sRejectReasonME, stPackRejectReasons.stPackCodesDBError.sMetsSearchCode) > 0 THEN
	sRejectReasonFSS := stPackRejectReasons.stPackCodesDBError.sFssSendCode;

ELSIF FIND(sRejectReasonME, stPackRejectReasons.stPackCodesBrandSpec.sMetsSearchCode) > 0 THEN
	sRejectReasonFSS := stPackRejectReasons.stPackCodesBrandSpec.sFssSendCode;

ELSE
	sRejectReasonFSS := stPackRejectReasons.stUnknownPackReject.sFssSendCode;
END_IF

F_PACK_GetRejectReasonFSS := sRejectReasonFSS;

END_FUNCTION

// ---- POUs/METS/Common LIB/01_PACK LIB/Pack Functions/F_PACK_HexToPackCode.TcPOU
FUNCTION F_PACK_HexToPackCode : STRING(255)
VAR_INPUT
	strPackCodeInHex		: STRING(255);
END_VAR
VAR

	nPackCodeLen		: INT;
	nCharIndex		: INT;
	strCharInHex			: STRING(2);
	nAsciiCode			:BYTE;
	strChar			: STRING(2);
END_VAR

(* reset output *)
F_PACK_HexToPackCode := '';

(* length of strPackCode *)
nPackCodeLen := LEN(strPackCodeInHex);

(* strPackCode contains data *)
IF nPackCodeLen > 0 THEN

	(* check each char in the code *)
	FOR nCharIndex := 1 TO nPackCodeLen BY 2 DO

		(* get char from string *)
		strCharInHex := MID(strPackCodeInHex, 2, nCharIndex);
		HEXSTR_TO_DATA(strCharInHex, ADR(nAsciiCode), SIZEOF(nAsciiCode));
		strChar := F_ToCHR(nAsciiCode);
		F_PACK_HexToPackCode := CONCAT(F_PACK_HexToPackCode, strChar);
	END_FOR
END_IF

END_FUNCTION

// ---- POUs/METS/Common LIB/01_PACK LIB/Pack Functions/F_PACK_ProgNumberMap.TcPOU
FUNCTION F_PACK_ProgNumberMap : BOOL

VAR
	nPackIndex			: INT;
END_VAR
(*All VAR_IN_OUT variables have been moved to the end of the declaration due to compatibility reasons*)
VAR_IN_OUT
	stImageData				: ST_SCANNER_ImageData;	(* scanner response data *)
END_VAR

(*Function used only for old type of camera porgram without ProgramNumber. Used only in clasic PAOL before Mx project.
All newer instalation should base on Progrmanumber for Code mapping*)

FOR nPackIndex := 1 TO LIMIT(1, stImageData.nCodesRead, cMAX_CAMERA_PROG_NUMBER)  DO

	IF stImageData.aCodeData[nPackIndex].nProgramNo = 0 THEN

		(* code is in upper left quadrant of image *)
		IF stImageData.aCodeData[nPackIndex].fXPos < 0 AND stImageData.aCodeData[nPackIndex].fYPos >= 0 THEN

			(* get pack position within Outer *)
			stImageData.aCodeData[nPackIndex].nProgramNo := 1;

		(* code is in lower left quadrant of image *)
		ELSIF stImageData.aCodeData[nPackIndex].fXPos < 0 AND stImageData.aCodeData[nPackIndex].fYPos < 0 THEN

			(* get pack position within Outer *)
			stImageData.aCodeData[nPackIndex].nProgramNo := 2;

		(* code is in upper right quadrant of image *)
		ELSIF stImageData.aCodeData[nPackIndex].fXPos >= 0 AND stImageData.aCodeData[nPackIndex].fYPos >= 0 THEN

			(* get pack position within Outer *)
			stImageData.aCodeData[nPackIndex].nProgramNo := 3;

		(* code is in lower right quadrant of image *)
		ELSIF stImageData.aCodeData[nPackIndex].fXPos >= 0 AND stImageData.aCodeData[nPackIndex].fYPos < 0 THEN

			(* get pack position within Outer *)
			stImageData.aCodeData[nPackIndex].nProgramNo := 4;
		END_IF
	END_IF
END_FOR

END_FUNCTION

// ---- POUs/METS/Common LIB/01_PACK LIB/Pack Functions/F_PACK_ValidateCodeASCII.TcPOU
FUNCTION F_PACK_ValidateCodeASCII : INT
VAR_INPUT
	strPackCode		: T_PACK_Barcode;
END_VAR
VAR
	nPackCodeLen	: INT;
	nCharIndex		: INT;
	strChar			: STRING(1);
END_VAR

(* reset output *)
F_PACK_ValidateCodeASCII := 0;

(* length of strPackCode *)
F_PACK_ValidateCodeASCII := LEN(strPackCode);

(* strPackCode contains data *)
IF nPackCodeLen > 0 THEN

	(* check each char in the code *)
	FOR nCharIndex := 1 TO nPackCodeLen DO

		(* get char from string *)
		strChar := MID(strPackCode, 1, nCharIndex);

		(* char is every alphanumeric char *)
		IF (F_ToASC(strChar) >= 16#21 AND  F_ToASC(strChar) <= 16#7A) THEN

			(* update valid char counter *)
			F_PACK_ValidateCodeASCII := F_PACK_ValidateCodeASCII + 1;
		END_IF
	END_FOR
END_IF

END_FUNCTION

// ---- POUs/METS/Common LIB/01_PACK LIB/Pack Functions/F_PACK_ValidateHexName.TcPOU
FUNCTION F_PACK_ValidateHexName : INT
VAR_INPUT
	strHexName		: STRING(255);
END_VAR
VAR
	nHexNameLen	: INT;
	nCharIndex		: INT;
	strChar			: STRING(1);
END_VAR

(* reset output *)
F_PACK_ValidateHexName := 0;

(* length of strPackCode *)
nHexNameLen := LEN(strHexName);

(* strPackCode contains data *)
IF nHexNameLen > 0 THEN

	(* check each char in the code *)
	FOR nCharIndex := 1 TO nHexNameLen DO

		(* get char from string *)
		strChar := MID(strHexName, 1, nCharIndex);

		(* char is every alphanumeric char *)
		IF (F_ToASC(strChar) >= 16#30 AND F_ToASC(strChar) <= 16#39) OR (F_ToASC(strChar) >= 16#41 AND F_ToASC(strChar) <= 16#46) THEN

			(* update valid char counter *)
			F_PACK_ValidateHexName := F_PACK_ValidateHexName + 1;
		END_IF
	END_FOR
END_IF

END_FUNCTION

// ---- POUs/METS/Common LIB/01_PACK LIB/Pack Functions/F_PACK_ValidateTimeStamp.TcPOU
FUNCTION F_PACK_ValidateTimeStamp : BOOL
VAR_INPUT
	sPack		: T_MaxString;
	stCTDateTime	: ST_SYSTEM_DateTime;
END_VAR
VAR
	sDateCode: STRING(8);
	nHour: INT;
	sDate: STRING(23);
END_VAR

(* reset output *)
F_PACK_ValidateTimeStamp := TRUE;

sDateCode := RIGHT(sPack, 8); (*now check entire 8 character datecode*)

IF  F_InvalidNumericChar(sDateCode) > 0 THEN
	F_PACK_ValidateTimeStamp := FALSE;
ELSE
	nHour := STRING_TO_INT(RIGHT(sDateCode, 2));
	IF nHour < 0 OR nHour > 23 THEN (*first check is to make sure no alphas are on the end*)
		F_PACK_ValidateTimeStamp := FALSE;
	ELSE
		sDate := CONCAT('20', LEFT(sDateCode, 2)); (*year*)
		sDate := F_CONCAT3(sDate, '-', MID(sDateCode, 2, 3)); (*month*)
		sDate := F_CONCAT3(sDate, '-', MID(sDateCode, 2, 5)); (*day**)
		sDate := F_CONCAT3(sDate, '-', RIGHT(sDateCode, 2)); (*hour*)
		sDate := CONCAT(sDate, ':00:00.000'); (*all the rest*)

		IF F_SYSTEM_DateCompare(STRING_TO_SYSTEMTIME(sDate), stCTDateTime.sSystemTime) > 0 THEN
			F_PACK_ValidateTimeStamp := FALSE;
		END_IF
	END_IF
END_IF

END_FUNCTION

// ---- POUs/METS/Common LIB/08_SOFTWARE LIB/String FBs/F_InvalidNumericChar.TcPOU
FUNCTION F_InvalidNumericChar : INT
VAR_INPUT
	sCode		: STRING(255);
END_VAR
VAR
	nCodeLen	: INT;
	nCharIndex		: INT;
	sChar			: STRING(1);
END_VAR

(* reset output *)
F_InvalidNumericChar := 0;

(* strPackCode contains data *)
IF LEN(sCode) > 0 THEN

	(* check each char in the code *)
	FOR nCharIndex := 1 TO LEN(sCode) DO

		(* get char from string *)
		sChar := MID(sCode, 1, nCharIndex);

		(* check if every char valid for proccessig*)
		IF (F_ToASC(sChar) < 16#30 OR  F_ToASC(sChar) >  16#39) THEN

			(* update valid char counter *)
			F_InvalidNumericChar := F_InvalidNumericChar + 1;
		END_IF
	END_FOR
END_IF

END_FUNCTION

// ---- POUs/METS/Common LIB/02_OUTER LIB/OAC FBs/FB_OAC_FindDB.TcPOU
(* converts strOuterBarcode to OAC filename and loads data *)
FUNCTION_BLOCK FB_OAC_FindDB
VAR_INPUT
	bExecute			: BOOL;		(* set TRUE to load OAC file *)
	sRetailSKU 			: T_CodeRSKU;
	sOuterBarcode		: T_MaxString;	(* Outer barcode *)
END_VAR
VAR_IN_OUT
	stOACDataDB					: ST_DB_OACDataCtrl;
	stCodeInfo_Outer			: ST_CodeInfo;
END_VAR
VAR_OUTPUT
	bDone				: BOOL;		(* TRUE = find file complete *)
	bBusy				: BOOL;		(* TRUE = find file in progress *)
	bError				: BOOL;		(* TRUE = error occurred *)
	nErrorID			: UDINT;	(* error code *)
	bOACDataFound		: BOOL;		(* TRUE = OAC file found *)
	bOACDataValid			: BOOL;
	stOACData			: ST_OAC_Data;	(* OAC data for strOuterBarcode *)
	sOACRecord		: T_MaxString;	(* OAC filename *)
	(*sOuterCodeAI		:T_MaxString;*)
END_VAR
VAR
	fbExecute			: R_TRIG;
	eState				: E_OAC_State;
	eErrorState				: E_OAC_State;
	eCodeAIType					: E_CodeAIType;

	tonTimeOut				: TON;
	rtTimeOutExec				: R_TRIG;
	
	stDiagOACDataDB					: ST_DB_OACDataCtrl;
	(*fbReadFile			: FB_XmlSrvRead;
	fbDecodeGS1				: FB_SCANNER_DecodeGS1;*)
END_VAR

(***************************************TimeOut *******************************************)
(* monitor Busy timeout *)
tonTimeOut( IN:=eState=E_OAC_DBREQUEST, PT:=cTHREE_SECONDS, Q=>);
(*	cTHREE_SECONDS						: TIME := T#3s;
	cFIVE_SECONDS						: TIME := t#5s;
	cTEN_SECONDS						: TIME := t#10s;*)

rtTimeOutExec(CLK:= tonTimeOut.Q);

IF rtTimeOutExec.Q THEN

	bError := TRUE;
	nErrorID := 100;
	eErrorState := eState;

	MEMSET(ADR(stOACDataDB), 16#00, SIZEOF(stOACDataDB));

	eState := E_OAC_DONE;
END_IF

(***************************************Execution*******************************************)

fbExecute(CLK := bExecute);

CASE eState OF

	(* idle *)
	E_OAC_IDLE:

		(* rising edge of bExecute *)
		IF fbExecute.Q = TRUE THEN

			(* initialise outputs *)
			bDone := FALSE;
			bBusy := TRUE;
			bError := FALSE;
			nErrorID := 0;
			sOACRecord := '';
			(* convert strOuterBarcode to OAC filename *)
			bOACDataFound := FALSE;
			bOACDataValid	:= FALSE;
			MEMSET(ADR(stOACData), 16#00, SIZEOF(stOACData));



			eState := E_OAC_DBREQUEST;

		ELSIF bExecute = FALSE THEN

			(* reset outputs *)
			bDone := FALSE;
			bBusy := FALSE;
			bError := FALSE;
			(*nErrorID := 0;*)

		END_IF

	E_OAC_DBREQUEST:

		stOACDataDB.bReadDataReq		:=TRUE;

		IF F_InvalidateASCIIChar(F_CODE_GetItem(sOuterBarcode, eCodeAIType.SerialCode, stCodeInfo_Outer)) >	0 	THEN

			stOACDataDB.sFileCodeName := '';
		ELSE
			stOACDataDB.sFileCodeName	:= F_CodeToHex(F_CODE_GetItem(sOuterBarcode , eCodeAIType.SerialCode, stCodeInfo_Outer));
		END_IF

		IF stOACDataDB.bDone THEN
			IF NOT stOACDataDB.bError THEN		(* f.ex not found, or DB transaction faild??*)

				stOACData := stOACDataDB.stOACStatusDB.stOACData;
				sOACRecord	:=  stOACDataDB.stOACStatusDB.stOACData.Barcode;
				(* OAC record exists *)
				bOACDataFound := TRUE;

				IF sRetailSKU = stOACData.RetailSKU  AND stOACData.OuterRejectCode = 'OK'    THEN
					(* OAC data is valid *)
					bOACDataValid := TRUE;
				END_IF
			ELSE
				bError := TRUE;
				nErrorID := stOACDataDB.nErrorID;

				eErrorState := eState;
			END_IF
			
			stDiagOACDataDB	:= stOACDataDB;
			MEMSET(ADR(stOACDataDB), 16#00, SIZEOF(stOACDataDB));

			eState := E_OAC_DONE;
		END_IF

	(* complete *)
	E_OAC_DONE:
		(* update outputs *)
		bDone := TRUE;
		bBusy := FALSE;

		eState := E_OAC_IDLE;


(* unknown state *)
ELSE

	eState := E_OAC_IDLE;

	(* clear outputs *)
	bDone := FALSE;
	bBusy := FALSE;
	bError := FALSE;
	(*nErrorID := 0;*)
	sOACRecord := '';
END_CASE

END_FUNCTION_BLOCK

// ---- POUs/METS/Common LIB/02_OUTER LIB/Outer FBs/FB_OUTER_ArchiveInvalidOuters.TcPOU
FUNCTION_BLOCK FB_OUTER_ArchiveInvalidOuters
VAR_INPUT
	_bUpdate:	BOOL;
	_bClearList: BOOL;
	_strReasonForReject:	STRING(255);
END_VAR
VAR_IN_OUT
	_aReasonForReject: ARRAY[0..50] OF STRING(255);
END_VAR
VAR
	rtrigExecute: R_TRIG;
END_VAR

rtrigExecute(CLK:= _bUpdate);

IF rtrigExecute.Q THEN
	MEMMOVE(ADR(_aReasonForReject[1]), ADR(_aReasonForReject[0]), SIZEOF(_aReasonForReject) - SIZEOF(_aReasonForReject[0]));
	_aReasonForReject[0] := _strReasonForReject;
END_IF

IF _bClearList THEN
	MEMSET(ADR(_aReasonForReject), 0, SIZEOF(_aReasonForReject));
END_IF

END_FUNCTION_BLOCK

// ---- POUs/METS/Common LIB/02_OUTER LIB/Outer FBs/FB_OUTER_CheckDuplicateStatus.TcPOU
(* Outer DMC status monitor *)
FUNCTION_BLOCK FB_OUTER_CheckDuplicateStatus
VAR_INPUT
	bExecute				: BOOL;			(* code scan done *)
	bReset			: BOOL;
	stImageData			: ST_SCANNER_ImageData;	(* image data structure *)
END_VAR
VAR_OUTPUT
	bDone				: BOOL;
	bLastBarcodeValid		: BOOL;			(* strLastBarcode is valid against strRetailSKU *)
	sLastBarcode			: STRING(255);		(* last barcode read *)
	nNoCodeFound		: INT;
	stLastImageData		: ST_SCANNER_ImageData;	(* image data structure *)
	tAveScanTime			: TIME;			(* average of last 10 scans *)
	bDuplicateAlarm		: BOOL;
END_VAR
VAR
	fbExecute			: R_TRIG;
	sSerialCode			: STRING(255);
	sPreviousBarcode		: STRING(255);

	tScanTime			: ARRAY[1..10] OF TIME;
	nMaxIndex			: INT;
	nScanValues			: INT;
	nIndex				: INT;
END_VAR

IF bReset THEN

	bLastBarcodeValid := FALSE;
	sLastBarcode := '';
	nNoCodeFound := 0;

	MEMSET(ADR(stLastImageData), 16#00, SIZEOF(stLastImageData));
END_IF

(* rising edge of bDone *)
fbExecute(CLK := bExecute);
IF fbExecute.Q = TRUE THEN
	bDone:= FALSE;
	bDuplicateAlarm := FALSE;

	(* log image data *)
	stLastImageData := stImageData;
	(* extract data string and status *)
	sLastBarcode := stLastImageData.aCodeData[1].strDataString;

	(* barcode found *)
	IF LEN(sLastBarcode) > 0 THEN
		bLastBarcodeValid := TRUE;

		IF sLastBarcode <> '' AND sLastBarcode = sPreviousBarcode THEN
			bDuplicateAlarm := TRUE;
		END_IF

		sPreviousBarcode := sLastBarcode;

		(* shifttScanTime array and add new tScanTime *)
		nMaxIndex := UDINT_TO_INT(SIZEOF(tScanTime) / SIZEOF(tScanTime[1]));
		MEMMOVE(ADR(tScanTime[2]), ADR(tScanTime[1]), SIZEOF(tScanTime) - SIZEOF(tScanTime[1]));
		tScanTime[1] := stLastImageData.tScanTime;
		nScanValues := LIMIT(1, nScanValues + 1, nMaxIndex);

		(* re-calculate average *)
		tAveScanTime := T#0ms;
		FOR nIndex := 1 TO nScanValues DO
			(* total scan time *)
			tAveScanTime := tAveScanTime + tScanTime[nIndex];
		END_FOR

		(* average scan time *)
		tAveScanTime := tAveScanTime / nScanValues;
	(* no code found *)
	ELSE
		(* reset Valid flag *)
		bLastBarcodeValid := FALSE;
		nNoCodeFound := nNoCodeFound + 1;
	END_IF
	bDone:= TRUE;
ELSE

	bDone:= FALSE;
	bDuplicateAlarm := FALSE;

END_IF

END_FUNCTION_BLOCK

// ---- POUs/METS/Common LIB/02_OUTER LIB/Outer FBs/FB_OUTER_FindErrorOuter.TcPOU
(* returns selected Outer for display in HMI, allows search for serial code in error Outers *)
FUNCTION_BLOCK FB_OUTER_FindErrorOuter
VAR_INPUT
	bErrorIndexPlus		: BOOL;		(* set TRUE to increment nErrorIndex *)
	bErrorIndexMinus		: BOOL;		(* set TRUE to decrement nErrorIndex *)
	bErrorUpdate			: BOOL;
	bEnableInvalidSearch	: BOOL;
	bClearData			: BOOL;			(* set TRUE to clear data for invalid Outers *)
	bSearchCode			: BOOL;		(* set TRUE to search for strSearchCode *)
	nStartIndex			: INT;		(* index to start search, allows searches for multiple matching codes *)
	arrErrorOuter			: ARRAY[1..cMAX_OUTER_STATUS_QUEUE] OF ST_OUTER_Status; (* status for last 50 failed Outers *)
	sProductInstruction		: ST_PCM_Status;
	bUseInterimCodeForValidation		: BOOL;
END_VAR
VAR_IN_OUT
	strSearchCode			: T_MaxString;	(* search code *)
	nErrorIndex			: INT;		(* index of Error Outer to be displayed *)
	stPackCodeInfo						: ST_CodeInfo;
	stOuterCodeInfo						: ST_CodeInfo;
	stOuterRejectReasons		: ST_RejectReasonsForOuter;
	bEnableRefeedButton	: BOOL;
	stFailureDiagnostic			: ST_HMI_OuterStatus;
END_VAR
VAR_OUTPUT
	bDone				: BOOL;		(* TRUE = search complete *)
	bBusy				: BOOL;		(* TRUE = search in progress *)
	bError				: BOOL;		(* TRUE = nFirstIndex out of range *)
	nErrorID				: UDINT;	(* error code *)
	bSearchCodeFound		: BOOL;		(* TRUE = Outer with strSearchCode found *)
	bErrorIndexChanged		: BOOL;
	bEnableRefeed			: BOOL;
	stErrorOuter			: ST_OUTER_Status; (* Outer for display *)
	strLastSerachCode		: T_MaxString;
END_VAR
VAR
	eCodeAIType				: E_CodeAIType;
	fbErrorIndexPlus		: R_TRIG;
	fbErrorIndexMinus		: R_TRIG;
	fbErrorUpdate			: R_TRIG;
	fbClearData			: R_TRIG;

	counter1 : INT;

	nMaxOuterIndex		: INT;
	nLastErrorIndex		: INT;

	eState				: E_OUTER_State;
	fbSearchCode			: R_TRIG;
	nMaxPackIndex		: INT;
	nSearchCodeLen		: INT;

	nOuterIndex			: INT;
	nPackIndex			: INT;
	strSerialCode			: T_MaxString;
	strSerialCode2			: T_MaxString;

	nGoodPackReads		: INT;

	nErrorIndexLocal		: INT;
	nSourceIndex			: INT;
	nRestorePackIndex		: INT;

END_VAR

(* rising edge on bErrorIndexPlus and bErrorIndexMinus *)
fbErrorIndexPlus(CLK := bErrorIndexPlus);
fbErrorIndexMinus(CLK := bErrorIndexMinus);
fbErrorUpdate(CLK := bErrorUpdate);

fbClearData(CLK := bClearData);

bErrorIndexChanged := FALSE;
nErrorIndexLocal := nErrorIndex;

(* max number of Outers and PacksPerOuter *)
nMaxOuterIndex := UDINT_TO_INT(SIZEOF(arrErrorOuter) / SIZEOF(arrErrorOuter[1]));
nMaxPackIndex := UDINT_TO_INT(SIZEOF(arrErrorOuter[1].stOACData.PackCode) / SIZEOF(arrErrorOuter[1].stOACData.PackCode[1]));

IF fbClearData.Q = TRUE THEN

	(* clear Outer error data *)
	MEMSET(ADR(stErrorOuter), 16#00, SIZEOF(stErrorOuter));
	nErrorIndex := 1;
END_IF

(* next error index *)
IF fbErrorIndexPlus.Q = TRUE THEN

	(* max number of Outers *)
	(*nMaxOuterIndex := UDINT_TO_INT(SIZEOF(arrErrorOuter) / SIZEOF(arrErrorOuter[1]));*)

	(* roll-over required *)
	IF nErrorIndex >= nMaxOuterIndex THEN

		(* roll-over to 1 *)
		nErrorIndex := 1;

	(* roll-over not required *)
	ELSE

		(* increment nErrorIndex *)
		nErrorIndex := nErrorIndex + 1;
	END_IF

(* previous error index *)
ELSIF fbErrorIndexMinus.Q = TRUE THEN

	(* max number of Outers *)
	(*nMaxOuterIndex := UDINT_TO_INT(SIZEOF(arrErrorOuter) / SIZEOF(arrErrorOuter[1]));*)

	(* roll-under required *)
	IF nErrorIndex <= 1 THEN

		(* roll-under to nMaxOuterIndex *)
		nErrorIndex := nMaxOuterIndex;

	(* roll-under not required *)
	ELSE

		(* decrement nErrorIndex *)
		nErrorIndex := nErrorIndex - 1;
	END_IF
END_IF

(* nErrorIndex is 0 *)
IF nErrorIndex = 0 THEN

	(* reset nErrorIndex and clear sErrorOuter *)
	MEMSET(ADR(stErrorOuter),16#00, SIZEOF(stErrorOuter));
	nErrorIndex := 1;

	bSearchCodeFound := FALSE;
	bEnableRefeedButton := FALSE;

(* nErrorIndex has changed *)
ELSIF nErrorIndex <> nLastErrorIndex  THEN
	(* nErrorIndex is valid *)
	IF nErrorIndex >= 1 AND nErrorIndex <= nMaxOuterIndex THEN

		(* move data for selected Outer to sErrorOuter *)
		MEMMOVE(ADR(stErrorOuter), ADR(arrErrorOuter[nErrorIndex]), SIZEOF(stErrorOuter));
		IF stErrorOuter.stOACData.Barcode = stErrorOuter.stOACData.AggregationCodes[1] AND stErrorOuter.stOACData.OuterRejectCode = stOuterRejectReasons.stOuterBarcodeNotRead.sMetsDisplayCode  THEN
			stErrorOuter.stOACData.Barcode := '';
		END_IF

		bSearchCodeFound := FALSE;
		bEnableRefeedButton := FALSE;

	(* nErrorIndex is valid *)
	ELSE
		(* reset nErrorIndex and clear sErrorOuter *)
		MEMSET(ADR(stErrorOuter),16#00, SIZEOF(stErrorOuter));
		nErrorIndex := 1;

		bSearchCodeFound := FALSE;
		bEnableRefeedButton := FALSE;
	END_IF

	bErrorIndexChanged := TRUE;
	counter1 := counter1+1;

	(* log last error index used *)
	nLastErrorIndex := nErrorIndex;

(* nErrorIndex has changed *)
ELSIF fbErrorUpdate.Q THEN

		(* move data for selected Outer to sErrorOuter *)
		MEMMOVE(ADR(stErrorOuter), ADR(arrErrorOuter[nErrorIndex]), SIZEOF(stErrorOuter));
		IF stErrorOuter.stOACData.Barcode = stErrorOuter.stOACData.AggregationCodes[1] AND stErrorOuter.stOACData.OuterRejectCode = stOuterRejectReasons.stOuterBarcodeNotRead.sMetsDisplayCode  THEN
			stErrorOuter.stOACData.Barcode := '';
		END_IF
END_IF

IF NOT bEnableInvalidSearch THEN
	bEnableRefeedButton := FALSE;
END_IF

(* monitor bSearchCode for rising edge *)
fbSearchCode(CLK := bSearchCode);

CASE eState OF

	(* idle *)
	E_OUTER_IDLE:

		(* rising edge of bSearchCode *)
		IF fbSearchCode.Q = TRUE THEN

			(* initialise outputs *)
			bDone := FALSE;
			bBusy := TRUE;
			bError := FALSE;
			nErrorID := 0;

			(* max number of Outers and PacksPerOuter *)
			(*nMaxOuterIndex := UDINT_TO_INT(SIZEOF(arrErrorOuter) / SIZEOF(arrErrorOuter[1]));
			nMaxPackIndex := UDINT_TO_INT(SIZEOF(arrErrorOuter[1].stOACData.PackCode) / SIZEOF(arrErrorOuter[1].stOACData.PackCode[1]));*)

			(* initialise vars *)
			bSearchCodeFound := FALSE;
			bEnableRefeed := FALSE;

			strLastSerachCode := strSearchCode;
			(* nStartIndex is valid *)
			IF nStartIndex >= 1 AND nStartIndex <= nMaxOuterIndex THEN

				(* 1st Outer to check *)
				nOuterIndex := nStartIndex;

				(* capitalise strSearchCode and calculate code length *)
				(*strSearchCode := F_ToUCase(strSearchCode);*)
				nSearchCodeLen := LEN(strSearchCode);

				eState := E_OUTER_SCAN;

			(* nFirstIndex is invalid *)
			ELSE

				(* update outputs *)
				bError := TRUE;
				nErrorID := 1;

				eState := E_OUTER_DONE;
			END_IF

		(* bSearchCode has been reset or strSearchCode has been cleared *)
		ELSIF bSearchCode = FALSE OR strSearchCode = '' THEN

			(* reset outputs *)
			bDone := FALSE;
			bBusy := FALSE;
			bError := FALSE;
			nErrorID := 0;
			bSearchCodeFound := FALSE;
			bEnableRefeed := FALSE;

		END_IF


	(* search for PackCode *)
	E_OUTER_SCAN:

		(* reset flag *)
		bSearchCodeFound := FALSE;
		bEnableRefeedButton := FALSE;
		nSourceIndex := 0;

		(* extract Outer serial code *)
		(*strSerialCode :=  F_CODE_GetItem(arrErrorOuter[nOuterIndex].stOACData.Barcode, eCodeAIType.SerialCode, stMachineConfig.stCodeInfo_Outer);*)

		(* check Outer serial code *)
		(*IF LEFT(strSerialCode, nSearchCodeLen) = strSearchCode THEN*)
		IF( strSearchCode = F_CODE_GetItem(arrErrorOuter[nOuterIndex].stOACData.Barcode, eCodeAIType.SerialCode, stOuterCodeInfo) )  OR
			(strSearchCode = arrErrorOuter[nOuterIndex].stOACData.AggregationCodes[1]  AND bUseInterimCodeForValidation) THEN

			(* strSearchCode found *)
			bSearchCodeFound := TRUE;
		(* check Pack codes *)
		ELSE

			(* for each Pack in Outer *)
			FOR nPackIndex := 1 TO nMaxPackIndex DO

				(* check for matching pack code *)
				(*IF LEFT(arrErrorOuter[nOuterIndex].stOACData.PackCode[nPackIndex], nSearchCodeLen) = strSearchCode THEN*)

				(*strSerialCode2 := F_CODE_GetItem(arrErrorOuter[nOuterIndex].stOACData.PackCode[nPackIndex], eCodeAIType.SerialCode, stMachineConfig.stCodeInfo_Pack);

				IF LEFT(strSerialCode2, nSearchCodeLen) = strSearchCode THEN*)
				IF strSearchCode = F_CODE_GetItem(arrErrorOuter[nOuterIndex].stOACData.PackCode[nPackIndex], eCodeAIType.SerialCode, stPackCodeInfo) THEN

					(* strSearchCode found *)
					bSearchCodeFound := TRUE;

					IF sProductInstruction.nPacksPerOuter - arrErrorOuter[nOuterIndex].stOACData.NumberOfLinkedPacks = 1 THEN

						FOR nRestorePackIndex := 1 TO sProductInstruction.nPacksPerOuter BY 1 DO

							IF arrErrorOuter[nOuterIndex].aOACPackStatus[nRestorePackIndex] = 0 OR arrErrorOuter[nOuterIndex].aOACPackStatus[nRestorePackIndex] = 1 THEN

									nSourceIndex := nRestorePackIndex;
								EXIT;
							END_IF

						END_FOR

						IF nSourceIndex > 0 THEN
							bEnableRefeedButton := TRUE;
						END_IF

					END_IF

					EXIT;
				END_IF
			END_FOR
		END_IF

		(* strSearchCode found *)
		IF bSearchCodeFound = TRUE THEN

			(* update indexes *)
			nErrorIndex := LIMIT(1, nOuterIndex, nMaxOuterIndex);
			nLastErrorIndex := nErrorIndex;

			bErrorIndexChanged := TRUE;

			(* move data for selected Outer to sErrorOuter *)
			MEMMOVE(ADR(stErrorOuter), ADR(arrErrorOuter[nErrorIndex]), SIZEOF(stErrorOuter));

			IF stErrorOuter.stOACData.Barcode = stErrorOuter.stOACData.AggregationCodes[1] AND stErrorOuter.stOACData.OuterRejectCode = stOuterRejectReasons.stOuterBarcodeNotRead.sMetsDisplayCode  THEN
				stErrorOuter.stOACData.Barcode := '';
			END_IF

			eState := E_OUTER_DONE;

		(* strSearchCode not found, more Outers to check *)
		ELSIF nOuterIndex < nMaxOuterIndex THEN

			(* next Outer *)
			nOuterIndex := nOuterIndex + 1;

		(* all Outers checked *)
		ELSE
			bEnableRefeed := TRUE;
			eState := E_OUTER_DONE;
		END_IF


	(* complete *)
	E_OUTER_DONE:

		(* update outputs *)
		bDone := TRUE;
		bBusy := FALSE;

		eState := E_OUTER_IDLE;


(* unknown state *)
ELSE

	eState := E_OUTER_IDLE;

	(* reset outputs *)
	bDone := TRUE;
	bBusy := FALSE;
	bError := TRUE;
	nErrorID := 16#FFFFFFFF;
	bSearchCodeFound := FALSE;
	bEnableRefeed := FALSE;
	bEnableRefeedButton := FALSE;
	MEMSET(ADR(stErrorOuter),16#00, SIZEOF(stErrorOuter));
END_CASE

IF fbErrorIndexPlus.Q OR fbErrorIndexMinus.Q OR fbErrorUpdate.Q OR bSearchCodeFound THEN

	IF stErrorOuter.stOACData.NumberOfLinkedPacks > 0 THEN
		nGoodPackReads := 0;
		FOR nPackIndex := 1 TO stErrorOuter.stOACData.NumberOfPacks DO
			IF stErrorOuter.aOACPackStatus[nPackIndex] > 4 AND stErrorOuter.stOACData.PackRejectID[nPackIndex] =0 THEN
				nGoodPackReads := nGoodPackReads + 1;
			END_IF
		END_FOR
	ELSE
		nGoodPackReads := 0;
	END_IF

	stFailureDiagnostic.sBarcode	:= stErrorOuter.stOACData.Barcode;

	MEMMOVE(ADR(stFailureDiagnostic.aAggregationCodes), ADR(stErrorOuter.stOACData.AggregationCodes), SIZEOF(stErrorOuter.stOACData.AggregationCodes));
	
	MEMMOVE(ADR(stFailureDiagnostic.aPackRejectCode), ADR(stErrorOuter.stOACData.PackRejectCode), SIZEOF(stErrorOuter.stOACData.PackRejectCode));
	MEMMOVE(ADR(stFailureDiagnostic.aPackRejectID), ADR(stErrorOuter.stOACData.PackRejectID), SIZEOF(stErrorOuter.stOACData.PackRejectID));
	
	stFailureDiagnostic.sProductionDate 	:= 	stErrorOuter.stOACData.ProductionDate;
	stFailureDiagnostic.sProductionTime	:=	stErrorOuter.stOACData.ProductionTime;
	
	stFailureDiagnostic.sOuterRejectCode		:= stErrorOuter.stOACData.OuterRejectCode;
	stFailureDiagnostic.nOuterRejectID		:= stErrorOuter.stOACData.OuterRejectID;

	MEMMOVE(ADR(stFailureDiagnostic.aPackCode), ADR(stErrorOuter.stOACData.PackCode), SIZEOF(stErrorOuter.stOACData.PackCode));
	MEMMOVE(ADR(stFailureDiagnostic.aOACPackStatus), ADR(stErrorOuter.aOACPackStatus), SIZEOF(stErrorOuter.aOACPackStatus));
	
	stFailureDiagnostic.nNumberOfPacks			:=	stErrorOuter.stOACData.NumberOfPacks;
	stFailureDiagnostic.nAcceptanceLevel			:=	stErrorOuter.stOACData.AcceptanceLevel;
	stFailureDiagnostic.nNumberOfLinkedPacks	:=	nGoodPackReads;
END_IF

END_FUNCTION_BLOCK

// ---- POUs/METS/Common LIB/02_OUTER LIB/Outer FBs/FB_OUTER_InterimCameraOut.TcPOU
FUNCTION_BLOCK FB_OUTER_InterimCameraOut
VAR_INPUT
	bFrontConfirmationCameraInUse	: BOOL;
	bCameraTrigger				: BOOL;
	bLightTrigger					: BOOL;
END_VAR
VAR_OUTPUT
	bRearScannerOut				: BOOL;
	bRearLightOut				: BOOL;
	bFrontScannerOut				: BOOL;
	bFrontLightOut				: BOOL;
END_VAR

IF  bFrontConfirmationCameraInUse THEN

	bFrontScannerOut := bCameraTrigger;
	bFrontLightOut := bLightTrigger;
ELSE

	bRearScannerOut := bCameraTrigger;
	bRearLightOut := bLightTrigger;
END_IF

END_FUNCTION_BLOCK

// ---- POUs/METS/Common LIB/02_OUTER LIB/Outer FBs/FB_OUTER_MasterListUpdate.TcPOU
FUNCTION_BLOCK FB_OUTER_MasterListUpdate
VAR_INPUT
	bUdateMasterList				: BOOL;
	bRejectCurrentOuter			: BOOL;

	sCurrentBarcodeRead			: T_MaxString;
END_VAR
VAR_OUTPUT
	aMasterList			: ARRAY[0..cMAX_OUTER_STATUS_QUEUE] OF T_MaxString;
	sCurrentBarcodeAdded	: T_MaxString;
END_VAR
VAR
	rtrigUpdateMasterlist	: R_TRIG;
END_VAR

rtrigUpdateMasterlist(CLK:=  bUdateMasterList AND NOT bRejectCurrentOuter);
IF rtrigUpdateMasterlist.Q THEN
	MEMMOVE(ADR(aMasterList[1]), ADR(aMasterList[0]), SIZEOF(aMasterList) - SIZEOF(aMasterList[0]));
	aMasterList[0] := sCurrentBarcodeRead;
	sCurrentBarcodeAdded := sCurrentBarcodeRead;
END_IF

END_FUNCTION_BLOCK

// ---- POUs/METS/Common LIB/02_OUTER LIB/Outer FBs/FB_OUTER_MoveOuterStatus.TcPOU
(* move Outer Status register [1..49] to [2..50] and clear Outer Status register [1]*)
FUNCTION_BLOCK FB_OUTER_MoveOuterStatus
VAR_INPUT
	_bExecute			: BOOL;
END_VAR
VAR_IN_OUT
	_aOuterStatus		: ARRAY[1..cMAX_OUTER_STATUS_QUEUE] OF ST_OUTER_Status;	(* Outer status register *)
END_VAR
VAR_OUTPUT
	bDone			: BOOL;			(* TRUE = complete *)
END_VAR
VAR
	fbExecute			: R_TRIG;
END_VAR

(* rising edge of bExecute *)
fbExecute(CLK:= _bExecute);

(* move CaseData *)
IF fbExecute.Q = TRUE THEN

	(* move Outer Status register [1..49] to [2..50] and clear Outer Status register [1]*)
	MEMMOVE(ADR(_aOuterStatus[2]), ADR(_aOuterStatus[1]), SIZEOF(_aOuterStatus) - SIZEOF(_aOuterStatus[1]));
	MEMSET(ADR(_aOuterStatus[1]), 16#00, SIZEOF(_aOuterStatus[1]));

	(* update output *)
	bDone := TRUE;

(* bExecute has been reset *)
ELSIF _bExecute = FALSE THEN

	(* clear output *)
	bDone := FALSE;
END_IF

END_FUNCTION_BLOCK

// ---- POUs/METS/Common LIB/02_OUTER LIB/Outer FBs/FB_OUTER_RepairOCVContentDB.TcPOU
FUNCTION_BLOCK FB_OUTER_RepairOCVContentDB
VAR_INPUT
	bExecute					: BOOL;			(* scan for completed Outer *)
	bResetErrorStats			: BOOL;
	stProductInstruction			: ST_PCM_Status;
	nPackPos1				: INT 	:=1;
	nPackPos2				: INT	:=2;
	bUseInterimCodeForValidation	: BOOL;
	stDuplicatedItem			: ST_RejectItems;(*stPackRejectReasons.stPackCodesDuplicated*)
	tTimeout					: TIME := t#1s;
END_VAR
VAR_IN_OUT
	sNewPackCodeRefeed		:T_PACK_Barcode;
	stPackCodeInfo						: ST_CodeInfo;
	aErrorOuters				: ARRAY[1..cMAX_OUTER_STATUS_QUEUE] OF ST_OUTER_Status;
	nErrorIndex				: INT;
	aOCVPackStatus			: ARRAY[1..cMAX_OUTER_STATUS_QUEUE] OF ST_OUTER_Status;
	stOCVDataDB					: ST_DB_OCVDataCtrl;
	stCodeInfo_Pack			: ST_CodeInfo;
	stCodeInfo_Intermediate		: ST_CodeInfo;
END_VAR
VAR_OUTPUT
	bDone					: BOOL;			(* TRUE = validation complete *)
	bBusy					: BOOL;			(* TRUE = validation in progress *)
	bError					: BOOL;			(* TRUE = validation error *)
	nErrorID					: UDINT;			(* error ID *)
	aOCVRecordDBName			 : ARRAY[1..2] OF T_MaxString;
	nOutersStoredInOCV		: UINT;
END_VAR
VAR
	fbExecute					: R_TRIG;
	eCodeAIType					: E_CodeAIType;
	
	tonTimeOut				: TON;
	rtTimeOutExec				: R_TRIG;
	eState					: E_OUTER_State;
	eErrorState				: E_OUTER_State;
	fbDuplicatesPackCodesDB		: FB_PACK_DuplicatesPackCodesDB;
	(*aOCVFileCodeName			: ARRAY[1..2] OF T_MaxString;
	fbWriteOCVFile			: FB_OCV_WriteFile;*)
	fbValidatePack				: FB_CODE_ValidateExplicitCode;

	stErrorOuterData			: ST_OUTER_Status;	(* Outer status array *)
	stEmptyOuterData			: ST_OUTER_Status;	(* Outer status array *)


	(*bAggregationCodes1Valid			: BOOL;
	bAggregationCodes2Valid			: BOOL;*)

	nPackIndex				: INT;
	nSourceIndex				: INT;

	nOuterIndex				: uINT;
	nMaxOuterIndex 			: UINT;
	bPackDataRemovedFromST	: BOOL;

	nStatusError				: UDINT;
	nValidationError			: UDINT;
	nEmptySource				: UDINT;

	nWriteOCVerror			: UDINT;
	sMemoPackCodeRefeed	:T_MaxString;

	(*Diagnostic counters*)
	aDiagCounter : ARRAY[0..5] OF INT;
	aDiagOCVDataDB				: ARRAY[0..1] OF ST_DB_OCVDataCtrl;

END_VAR

(***************************************TimeOut *******************************************)
(* monitor Busy timeout *)
tonTimeOut( IN:=bBusy, PT:=tTimeout, Q=>);

rtTimeOutExec(CLK:= tonTimeOut.Q);

IF rtTimeOutExec.Q THEN

	bError := TRUE;
	nErrorID := 10;
	sNewPackCodeRefeed := '';

	MEMSET(ADR(stOCVDataDB), 16#00, SIZEOF(stOCVDataDB));

	eState := E_OUTER_DONE;
END_IF

(***************************************Execution*******************************************)


(* monitor rising edge of bExecute *)
fbExecute(CLK := bExecute);

IF bResetErrorStats THEN

	(* clear error statistic counters *)
	nStatusError := 0;
	nValidationError := 0;
	nEmptySource := 0;
	nOutersStoredInOCV := 0;
	nWriteOCVerror := 0;
	sMemoPackCodeRefeed := '';
END_IF

(* rising edge of bExecute *)
CASE eState OF

	(* idle *)
	E_OUTER_IDLE:

		(* scan for completed Outer when OAC files are required *)
		IF fbExecute.Q = TRUE THEN

			(* update outputs *)
			bDone := FALSE;
			bBusy := TRUE;
			bError := FALSE;
			nErrorID := 0;

			aDiagCounter[0] := aDiagCounter[0] +1;

			eState := E_OUTER_SCAN;

		(* no action required *)
		ELSIF bExecute = FALSE THEN

			(* reset outputs *)
			bDone := FALSE;
			bBusy := FALSE;
			bError := FALSE;
			(*bAggregationCodes1Valid := FALSE;
			bAggregationCodes2Valid := FALSE;
			fbWriteOCVFile(bExecute := FALSE);
			nErrorID := 0;*)

		END_IF

	(* scan for completed Outer *)
	E_OUTER_SCAN:

		bBusy := TRUE;
		nSourceIndex := 0;
		stErrorOuterData := aErrorOuters[nErrorIndex];

		IF stProductInstruction.nPacksPerOuter - stErrorOuterData.stOACData.NumberOfLinkedPacks = 1  AND sNewPackCodeRefeed <> '' THEN

			FOR nPackIndex := 1 TO stProductInstruction.nPacksPerOuter BY 1 DO

				IF  stErrorOuterData.aOACPackStatus[nPackIndex] = 0 OR stErrorOuterData.aOACPackStatus[nPackIndex] = 1  THEN

						nSourceIndex := nPackIndex;
					EXIT;
				END_IF
			END_FOR
		END_IF


		IF nSourceIndex > 0 THEN

			aDiagCounter[1] := aDiagCounter[1] +1;

			fbValidatePack(	sFullCode := sNewPackCodeRefeed,
							stCodeInfo := stPackCodeInfo,
							stProductInstruction := stProductInstruction);


			IF fbValidatePack.bValidationOK THEN

				stErrorOuterData.stOACData.PackCode[nSourceIndex]:= sNewPackCodeRefeed;
				stErrorOuterData.stOACData.PackCodeStatus[nSourceIndex].6 := TRUE;

				aDiagCounter[2] := aDiagCounter[2] +1;

				(*fbChekcDupPackCode(nNumberPackInOuters := stProductInstruction.nPacksPerOuter,
							sOuterStatus := stErrorOuterData,
							stDuplicatedItem := stDuplicatedItem,
							bDuplicateFound => 	);*)

				fbDuplicatesPackCodesDB(
					stDuplicatedItem := stDuplicatedItem,
					bExtendedDupCheck	:=	FALSE,
					stOuterStatus := stErrorOuterData,
					stLastOuterStatus := stEmptyOuterData,
					bDuplicateFound =>
					);


				IF NOT stErrorOuterData.nStatus.23 (*AND NOT stErrorOuterData.nStatus.26*) THEN


					stErrorOuterData.aOACPackStatus[nSourceIndex]:= 5;
					stErrorOuterData.stOACData.PackRejectCode[nSourceIndex]:= 'OK';
					stErrorOuterData.stOACData.PackRejectID[nSourceIndex]	:= 0;

					IF nPackPos1= nSourceIndex AND stErrorOuterData.stOACData.AggregationCodes[1] = '' THEN stErrorOuterData.stOACData.AggregationCodes[1] := sNewPackCodeRefeed; END_IF
					IF nPackPos2= nSourceIndex AND stErrorOuterData.stOACData.AggregationCodes[2] = '' THEN stErrorOuterData.stOACData.AggregationCodes[2] := sNewPackCodeRefeed; END_IF

					stErrorOuterData.aPackCodes[nSourceIndex].sBuffer[1].strCode := stErrorOuterData.stOACData.PackCode[nSourceIndex];
					stErrorOuterData.aPackCodes[nSourceIndex].sBuffer[1].nStatus := stErrorOuterData.aOACPackStatus[nSourceIndex];
					stErrorOuterData.aPackCodes[nSourceIndex].sBuffer[1].nStringSize := LEN(stErrorOuterData.stOACData.PackCode[nSourceIndex]);
					stErrorOuterData.aPackCodes[nSourceIndex].sBuffer[2].strCode := stErrorOuterData.stOACData.PackCode[nSourceIndex];
					stErrorOuterData.aPackCodes[nSourceIndex].sBuffer[2].nStatus := stErrorOuterData.aOACPackStatus[nSourceIndex];
					stErrorOuterData.aPackCodes[nSourceIndex].sBuffer[2].nStringSize := LEN(stErrorOuterData.stOACData.PackCode[nSourceIndex]);

					stErrorOuterData.stOACData.NumberOfLinkedPacks := stProductInstruction.nPacksPerOuter;

					aDiagCounter[3] := aDiagCounter[3] +1;

					eState := E_OUTER_CHECKPACKS;
				ELSE
					stErrorOuterData.stOACData.PackCode[nSourceIndex]:= 'STATUS REJECTED';

					nStatusError := nStatusError+1;
					sNewPackCodeRefeed := '';
					bError := TRUE;
					nErrorID := 1;

					eState := E_OUTER_IDLE;
				END_IF
			ELSE
				stErrorOuterData.stOACData.PackCode[nSourceIndex]:= 'CODE INVALIDE';
				stErrorOuterData.aOACPackStatus[nSourceIndex]:= 2;

				nValidationError := nValidationError+1;
				sNewPackCodeRefeed := '';

				bError := TRUE;
				nErrorID := 2;


				eState := E_OUTER_IDLE;
			END_IF

		ELSE
			nEmptySource := nEmptySource+1;
			sNewPackCodeRefeed := '';

			bError := TRUE;
			nErrorID := 3;

			eState := E_OUTER_IDLE;
		END_IF

	E_OUTER_CHECKPACKS:

		nMaxOuterIndex := SIZEOF(aOCVPackStatus) / SIZEOF(aOCVPackStatus[1]);
		bPackDataRemovedFromST := FALSE;

		FOR nPackIndex := 1 TO stProductInstruction.nPacksPerOuter BY 1 DO
			IF nPackIndex  <> nSourceIndex  THEN
				FOR nOuterIndex := 1 TO nMaxOuterIndex BY 1 DO

					IF aOCVPackStatus[nOuterIndex].stOACData.PackCode[nPackIndex] = stErrorOuterData.stOACData.PackCode[nPackIndex] THEN

						MEMMOVE(ADR(aOCVPackStatus[nOuterIndex]), ADR(aOCVPackStatus[nOuterIndex + 1]), SIZEOF(aOCVPackStatus[1]) * (nMaxOuterIndex - nOuterIndex) );
						MEMSET(ADR(aOCVPackStatus[nMaxOuterIndex]), 0, SIZEOF(aOCVPackStatus[1]));
						bPackDataRemovedFromST := TRUE;
						EXIT;
					END_IF

				END_FOR
			END_IF
			IF bPackDataRemovedFromST THEN
				EXIT;
			END_IF
		END_FOR

		eState := E_OUTER_WRITEDATA;


	E_OUTER_WRITEDATA:

		IF F_InvalidateASCIIChar(F_CODE_GetItem(stErrorOuterData.stOACData.AggregationCodes[1]  , eCodeAIType.SerialCode, SEL(bUseInterimCodeForValidation, stCodeInfo_Pack, stCodeInfo_Intermediate))) >	0 	THEN

			stErrorOuterData.sDataSourceTracker  := 'AGG_INVAL';
			stErrorOuterData.nStatus.22 := TRUE;
		ELSE
			stOCVDataDB.sFileCodeName1	:= F_CodeToHex(F_CODE_GetItem(stErrorOuterData.stOACData.AggregationCodes[1]  , eCodeAIType.SerialCode, SEL(bUseInterimCodeForValidation, stCodeInfo_Pack, stCodeInfo_Intermediate)));
		END_IF

		IF F_InvalidateASCIIChar(F_CODE_GetItem(stErrorOuterData.stOACData.AggregationCodes[2] , eCodeAIType.SerialCode,   stCodeInfo_Pack)) >	0 	THEN

			stErrorOuterData.sDataSourceTracker  := 'AGG_INVAL';
			stErrorOuterData.nStatus.22 := TRUE;
		ELSE
			stOCVDataDB.sFileCodeName2	:= F_CodeToHex(F_CODE_GetItem(stErrorOuterData.stOACData.AggregationCodes[2] , eCodeAIType.SerialCode,   stCodeInfo_Pack)); (*no reason to have 2 diffrent intermediate codes*)
		END_IF

		stOCVDataDB.stOCVStatusDB	:= stErrorOuterData;
		stOCVDataDB.bCreateDataReq := TRUE;

(*Place for HectorDB block*)

		IF	stOCVDataDB.bDone	THEN

			aErrorOuters[nErrorIndex].aOACPackStatus[nSourceIndex]:= 6;

			aErrorOuters[nErrorIndex].stOACData.PackCode[nSourceIndex]:= sNewPackCodeRefeed;
			aErrorOuters[nErrorIndex].stOACData.PackRejectCode[nSourceIndex]:= 'OCV Restored';
			aErrorOuters[nErrorIndex].stOACData.PackRejectID[nSourceIndex]:= 0;

			aErrorOuters[nErrorIndex].stOACData.NumberOfLinkedPacks := stProductInstruction.nPacksPerOuter;
			aErrorOuters[nErrorIndex].stOACData.OuterRejectCode := CONCAT(aErrorOuters[nErrorIndex].stOACData.OuterRejectCode, ' *OCV Restored*');
			aErrorOuters[nErrorIndex].stOACData.OuterRejectID := 0;

			(* count OCV files written *)
			nOutersStoredInOCV := nOutersStoredInOCV + 1;
			aDiagCounter[5] := aDiagCounter[5] +1;

			aOCVRecordDBName[1] := stOCVDataDB.sFileCodeName1;
			aOCVRecordDBName[2] := stOCVDataDB.sFileCodeName2;

			IF NOT  stOCVDataDB.bError THEN
				(* update sOuterStatus - OCV file write error  - general error for OCV *)
				nWriteOCVerror := nWriteOCVerror +1;
			ELSE
				bError := TRUE;
				nErrorID := stOCVDataDB.nErrorID;

				sNewPackCodeRefeed := '';;
				eErrorState := eState;
			END_IF

			aDiagOCVDataDB[0]	:= stOCVDataDB;

			MEMSET(ADR(stOCVDataDB), 16#00, SIZEOF(stOCVDataDB));

			eState := E_OUTER_DONE;
		END_IF

	(* OCV file complete *)
	E_OUTER_DONE:

		sMemoPackCodeRefeed := sNewPackCodeRefeed;
		sNewPackCodeRefeed := '';

		(* update outputs *)
		bDone := TRUE;
		bBusy := FALSE;

		eState := E_OUTER_IDLE;

(* unknown state *)
ELSE
	eState := E_OUTER_IDLE;
END_CASE

END_FUNCTION_BLOCK

// ---- POUs/METS/Common LIB/02_OUTER LIB/Outer FBs/FB_OUTER_RestoreOCVDataFromStruct.TcPOU
(* scan for and validate Outers marked as requiring validation *)
FUNCTION_BLOCK FB_OUTER_RestoreOCVDataFromStruct
VAR_INPUT
	bExecute				: BOOL;			(* scan for completed Outer *)
	bEnableRestoreOCV		: BOOL;
	bReset				: BOOL;
END_VAR
VAR_IN_OUT
	arrOCVPackStatus		: ARRAY[1..cMAX_OUTER_STATUS_QUEUE] OF ST_OUTER_Status;	(* Outer status register - would be nice to call it PACK Status and remove unnecesary stuff*)
	arrOuterStatus			: ARRAY[1..cMAX_OUTER_STATUS_QUEUE] OF ST_OUTER_Status;	(* Outer status array *)
	sProductInstruction		: ST_PCM_Status;					(* Product Instruction *)
END_VAR
VAR_OUTPUT
	bDone				: BOOL;			(* TRUE = validation complete *)
	bBusy				: BOOL;			(* TRUE = validation in progress *)

	nOutersRestored		: UDINT;		(* Outers restored *)
	nOutersProcessed 		: UDINT;

END_VAR
VAR
	fbExecute				: R_TRIG;
	eState				: E_OUTER_State;

	sOuterStatus			: ST_OUTER_Status;	(* Outer status *)
	nMaxOuterIndex		: INT;
	nOuterIndex			: INT;
	nSourceIndex			: INT;

	nOuterIndex1			: INT;
	nOuterIndex2			: INT;

	nPrevOuterIndex		: INT;
	nNextOuterIndex		: INT;

	sPrevOuterStatus		: ST_OUTER_Status;
	sNextOuterStatus		: ST_OUTER_Status;

	(*aNullPackCode		: ARRAY[1..cMAX_PACKS_PER_OUTER] OF T_PACK_Barcode;*)
END_VAR

IF bReset THEN

	nOutersRestored		:= 0;
	nOutersProcessed 		:= 0;
END_IF

(* monitor rising edge of bExecute *)
fbExecute(CLK := bExecute);

(* rising edge of bExecute *)
CASE eState OF

	(* idle *)
	E_OUTER_IDLE:

		(* scan for completed Outers when validation is active *)
		IF fbExecute.Q = TRUE THEN

			(* update outputs *)
			bDone := FALSE;
			bBusy := TRUE;


			(* reset outputs *)

			(*nPrevOuterIndex 	:= 0;
			nNextOuterIndex 	:= 0;*)

			(* max Outer index *)
			nMaxOuterIndex := UDINT_TO_INT(SIZEOF(arrOuterStatus) / SIZEOF(arrOuterStatus[1]));
			(*nSourceIndex := 0;*)

			eState := E_OUTER_SCAN;

		(* no action required *)
		ELSIF bExecute = FALSE THEN

			(* reset outputs *)
			bDone := FALSE;
			bBusy := FALSE;

		END_IF


	(* scan for completed Outer *)
	E_OUTER_SCAN:

		(* preset target state, will be over-written if an Outer requiringvalidation is found *)
		eState := E_OUTER_DONE;

		(* initialise source index *)
		nSourceIndex 		:= 0;
		nPrevOuterIndex 	:= 0;
		nNextOuterIndex 	:= 0;

		(* reset Outers Structures *)
		MEMSET(ADR(sPrevOuterStatus), 16#00, SIZEOF(sPrevOuterStatus));
		MEMSET(ADR(sOuterStatus), 16#00, SIZEOF(sOuterStatus));
		MEMSET(ADR(sNextOuterStatus), 16#00, SIZEOF(sNextOuterStatus));

		IF bEnableRestoreOCV AND sProductInstruction.nOpMode = 11 THEN
			(* for each Outer in Outer Status array *)
			FOR nOuterIndex := nMaxOuterIndex  TO 2 BY -1  DO
				(* Outer data ready for validation and not marked as passed or failed *)
				IF arrOuterStatus[nOuterIndex].nStatus.9 AND  arrOuterStatus[nOuterIndex].nStatus.16  AND  arrOuterStatus[nOuterIndex].nStatus.17  THEN
					(* index of Outer to be processed *)
					nSourceIndex := nOuterIndex;
					EXIT;
				END_IF
			END_FOR
		END_IF

		(* Outer found that requires validation *)
		IF nSourceIndex > 2 THEN

			(* copy Outer data from Outer Status array and extract SerialCode *)
			sPrevOuterStatus	:= arrOuterStatus[nSourceIndex - 1];
			sOuterStatus		:= arrOuterStatus[nSourceIndex];
			sNextOuterStatus	:= arrOuterStatus[nSourceIndex + 1];

			nOutersProcessed 		:= nOutersProcessed 	+ 1;

			sOuterStatus.stOACData.DataSource		:= 'NO_R';
			sOuterStatus.nStatus.16 := FALSE;

			eState := E_OUTER_VALIDATE;
		END_IF


	(* restore OAC data *)
	E_OUTER_VALIDATE:

		FOR nOuterIndex1 := nMaxOuterIndex  TO 1 BY -1  DO

			(*IF MEMCMP(ADR(arrOCVPackStatus[nOuterIndex].stOACData.PackCode), ADR(sPrevOuterStatus.stOACData.PackCode), SIZEOF(sPrevOuterStatus.stOACData.PackCode)) = 0 	AND
				MEMCMP(ADR(sPrevOuterStatus.stOACData.PackCode), ADR(aNullPackCode), SIZEOF(sPrevOuterStatus.stOACData.PackCode)) <> 0 							THEN;
				nPrevOuterIndex := nOuterIndex;
			END_IF

			IF MEMCMP(ADR(arrOCVPackStatus[nOuterIndex].stOACData.PackCode), ADR(sNextOuterStatus.stOACData.PackCode), SIZEOF(sNextOuterStatus.stOACData.PackCode)) = 0 	AND
				MEMCMP(ADR(sNextOuterStatus.stOACData.PackCode), ADR(aNullPackCode) , SIZEOF(sNextOuterStatus.stOACData.PackCode)) <> 0 							THEN;

				nNextOuterIndex := nOuterIndex;
			END_IF*)

(*********************condition expilitly one by one - MEMCMP had non consistent behaviour with table of strng************************************************************************)

			IF arrOCVPackStatus[nOuterIndex1].stOACData.PackCode[1] = sPrevOuterStatus.stOACData.PackCode[1] 		AND
				arrOCVPackStatus[nOuterIndex1].stOACData.PackCode[2] = sPrevOuterStatus.stOACData.PackCode[2] 	AND
				arrOCVPackStatus[nOuterIndex1].stOACData.PackCode[3] = sPrevOuterStatus.stOACData.PackCode[3] 	AND
				arrOCVPackStatus[nOuterIndex1].stOACData.PackCode[4] = sPrevOuterStatus.stOACData.PackCode[4] 	AND
				arrOCVPackStatus[nOuterIndex1].stOACData.PackCode[5] = sPrevOuterStatus.stOACData.PackCode[5] 	AND
				arrOCVPackStatus[nOuterIndex1].stOACData.PackCode[6] = sPrevOuterStatus.stOACData.PackCode[6] 	AND
				arrOCVPackStatus[nOuterIndex1].stOACData.PackCode[7] = sPrevOuterStatus.stOACData.PackCode[7] 	AND
				arrOCVPackStatus[nOuterIndex1].stOACData.PackCode[8] = sPrevOuterStatus.stOACData.PackCode[8] 	AND
				arrOCVPackStatus[nOuterIndex1].stOACData.PackCode[9] = sPrevOuterStatus.stOACData.PackCode[9] 	AND
 				arrOCVPackStatus[nOuterIndex1].stOACData.PackCode[10] = sPrevOuterStatus.stOACData.PackCode[10]	AND
				sPrevOuterStatus.stOACData.NumberOfLinkedPacks > 0										THEN

				nPrevOuterIndex := nOuterIndex1;
				EXIT;
			END_IF
		END_FOR

		FOR nOuterIndex2 := nMaxOuterIndex  TO 1 BY -1  DO
			IF arrOCVPackStatus[nOuterIndex2].stOACData.PackCode[1] = sNextOuterStatus.stOACData.PackCode[1] 		AND
				arrOCVPackStatus[nOuterIndex2].stOACData.PackCode[2] = sNextOuterStatus.stOACData.PackCode[2] 	AND
				arrOCVPackStatus[nOuterIndex2].stOACData.PackCode[3] = sNextOuterStatus.stOACData.PackCode[3] 	AND
				arrOCVPackStatus[nOuterIndex2].stOACData.PackCode[4] = sNextOuterStatus.stOACData.PackCode[4] 	AND
				arrOCVPackStatus[nOuterIndex2].stOACData.PackCode[5] = sNextOuterStatus.stOACData.PackCode[5] 	AND
				arrOCVPackStatus[nOuterIndex2].stOACData.PackCode[6] = sNextOuterStatus.stOACData.PackCode[6] 	AND
				arrOCVPackStatus[nOuterIndex2].stOACData.PackCode[7] = sNextOuterStatus.stOACData.PackCode[7] 	AND
				arrOCVPackStatus[nOuterIndex2].stOACData.PackCode[8] = sNextOuterStatus.stOACData.PackCode[8] 	AND
				arrOCVPackStatus[nOuterIndex2].stOACData.PackCode[9] = sNextOuterStatus.stOACData.PackCode[9] 	AND
 				arrOCVPackStatus[nOuterIndex2].stOACData.PackCode[10] = sNextOuterStatus.stOACData.PackCode[10]	AND
				sNextOuterStatus.stOACData.NumberOfLinkedPacks > 0										THEN

				nNextOuterIndex := nOuterIndex2;
				EXIT;
			END_IF
		END_FOR

		IF nPrevOuterIndex > 0 AND nNextOuterIndex > 0 THEN
			IF nNextOuterIndex - nPrevOuterIndex = 2 THEN

				sOuterStatus.aOACPackStatus				 := arrOCVPackStatus[nPrevOuterIndex + 1].aOACPackStatus;
				sOuterStatus.aPackCodes						:= arrOCVPackStatus[nPrevOuterIndex + 1].aPackCodes;

				sOuterStatus.stOACData.AggregationCodes[1]			:= 'RESTORED';
				sOuterStatus.stOACData.AggregationCodes[2]			:= 'RESTORED';


				sOuterStatus.stOACData.NumberOfLinkedPacks 	:= arrOCVPackStatus[nPrevOuterIndex + 1].stOACData.NumberOfLinkedPacks;
				sOuterStatus.stOACData.PackCode				:= arrOCVPackStatus[nPrevOuterIndex + 1].stOACData.PackCode;
				sOuterStatus.stOACData.PackRejectCode 			:= arrOCVPackStatus[nPrevOuterIndex + 1].stOACData.PackRejectCode;
				sOuterStatus.stOACData.PackRejectID 			:= arrOCVPackStatus[nPrevOuterIndex + 1].stOACData.PackRejectID;
				sOuterStatus.stOACData.PackTimeStamp 			:= arrOCVPackStatus[nPrevOuterIndex + 1].stOACData.PackTimeStamp;
				sOuterStatus.stOACData.DataSource		:= 'REST';

				nOutersRestored 		:= nOutersRestored 	+ 1;
				sOuterStatus.nStatus.17	:= TRUE;

			END_IF
		END_IF

		eState := E_OUTER_STATUS;

	(* update Outer status *)
	E_OUTER_STATUS:


		(* move sOuterStatus data back to shift reg *)
		FOR nOuterIndex := 1 TO nMaxOuterIndex DO

			(* matching nTriggerID found *)
			IF arrOuterStatus[nOuterIndex].nTriggerID = sOuterStatus.nTriggerID THEN

				(* move updated Outer data to shift reg *)
				arrOuterStatus[nOuterIndex] := sOuterStatus;

				EXIT;
			END_IF
		END_FOR

		eState := E_OUTER_SCAN;


	(* OAC file complete *)
	E_OUTER_DONE:

		(* update outputs *)
		bDone := TRUE;
		bBusy := FALSE;

		eState := E_OUTER_IDLE;


(* unknown state *)
ELSE

	eState := E_OUTER_IDLE;
END_CASE

END_FUNCTION_BLOCK

// ---- POUs/METS/Common LIB/02_OUTER LIB/Outer FBs/FB_OUTER_ShiftConfimrCodeQ.TcPOU
FUNCTION_BLOCK FB_OUTER_ShiftConfimrCodeQ
VAR_INPUT
	bClearPackConfirmationQueue	: BOOL;
	stConfirmationBarcode		: ST_SCANNER_ImageData;	(* 2D barcode from scanner *)
	bSensor1				: BOOL;
	bSensor2				: BOOL;
	bSensor3				: BOOL;
	bSensor4				: BOOL;
	stCodeInfo_Pack						: ST_CodeInfo;
END_VAR
VAR_IN_OUT
	stPackConfirmationQueue	: ST_PACK_ConfirmationQueue;
END_VAR
VAR_OUTPUT
	stInterimBarcodeForLabeler	: ST_SCANNER_ImageData;
	stAggregationBarcode		: ST_SCANNER_ImageData;
END_VAR
VAR
	fbExecute1			: R_TRIG;
	fbExecute2			: R_TRIG;
	fbExecute3			: R_TRIG;
	fbExecute4			: R_TRIG;

	bEnableSesnor2		: BOOL;
	bEnableSesnor3		: BOOL;

	nQueueIndex		: INT;
	nMaxQueueIndex	: INT;

	fbDebugCNT							: FB_DEBUG_CounterArray;
	aCNTDebug							: ARRAY [1..10] OF UDINT;
	bResetCNT							: BOOL;

END_VAR

IF bClearPackConfirmationQueue THEN
	MEMSET(ADR(stPackConfirmationQueue), 16#00, SIZEOF(stPackConfirmationQueue));
	MEMSET(ADR(stAggregationBarcode), 16#00, SIZEOF(stAggregationBarcode));
END_IF
(* rising edge OF bExecute *)
fbExecute1(CLK:= bSensor1);
fbExecute2(CLK:= bSensor2);
fbExecute3(CLK:= bSensor3);
fbExecute4(CLK:= bSensor4);

Debug();

(* add Outer to sInfeedQueue *)
IF fbExecute1.Q THEN

	stPackConfirmationQueue.aPackQueue[1]:= stConfirmationBarcode;
	stPackConfirmationQueue.nIndex := stPackConfirmationQueue.nIndex + 1;
	bEnableSesnor2 := TRUE;
END_IF

IF fbExecute2.Q AND bEnableSesnor2 THEN

	bEnableSesnor2 := FALSE;
	stPackConfirmationQueue.aPackQueue[2]:= stPackConfirmationQueue.aPackQueue[1];
	stInterimBarcodeForLabeler := stPackConfirmationQueue.aPackQueue[2];
	MEMSET(ADR(stPackConfirmationQueue.aPackQueue[1]), 16#00, SIZEOF(stPackConfirmationQueue.aPackQueue[1	]));
	bEnableSesnor3 := TRUE;

END_IF

IF fbExecute3.Q AND bEnableSesnor3 THEN
	bEnableSesnor3 := FALSE;
	stPackConfirmationQueue.aPackQueue[3]:= stPackConfirmationQueue.aPackQueue[2];
	stAggregationBarcode :=  stPackConfirmationQueue.aPackQueue[3];
	MEMSET(ADR(stPackConfirmationQueue.aPackQueue[2]), 16#00, SIZEOF(stPackConfirmationQueue.aPackQueue[2	]));

END_IF


IF fbExecute4.Q THEN
	MEMSET(ADR(stPackConfirmationQueue.aPackQueue[3]), 16#00, SIZEOF(stPackConfirmationQueue.aPackQueue[3	]));
	stPackConfirmationQueue.nIndex := stPackConfirmationQueue.nIndex- 1;

END_IF

ACTION Debug:
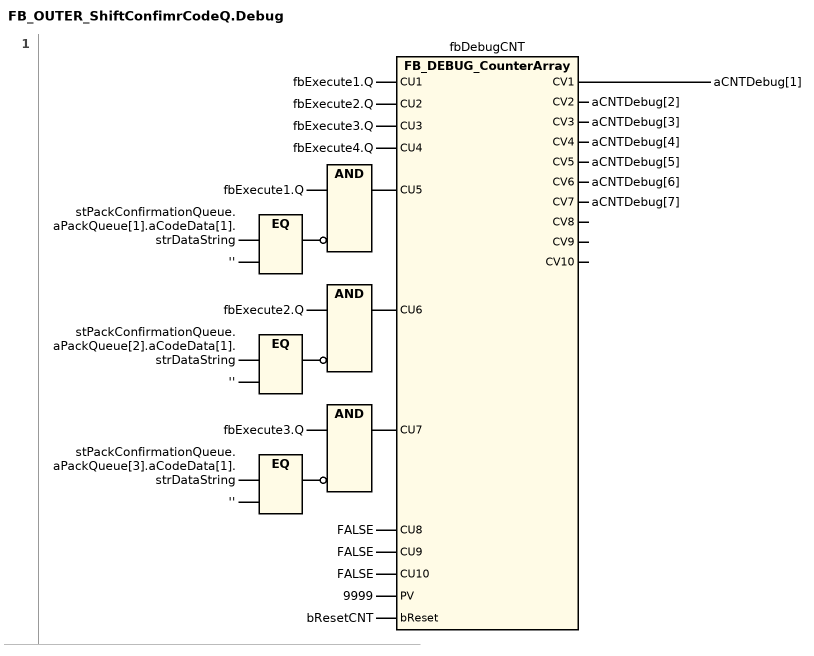
// NETWORK 1
fbDebugCNT(
    CU1 := fbExecute1.Q,
    CU2 := fbExecute2.Q,
    CU3 := fbExecute3.Q,
    CU4 := fbExecute4.Q,
    CU5 := fbExecute1.Q AND NOT (stPackConfirmationQueue.aPackQueue[1].aCodeData[1].strDataString = ''),
    CU6 := fbExecute2.Q AND NOT (stPackConfirmationQueue.aPackQueue[2].aCodeData[1].strDataString = ''),
    CU7 := fbExecute3.Q AND NOT (stPackConfirmationQueue.aPackQueue[3].aCodeData[1].strDataString = ''),
    CU8 := FALSE,
    CU9 := FALSE,
    CU10 := FALSE,
    PV := 9999,
    bReset := bResetCNT,
    CV2 => aCNTDebug[2],
    CV3 => aCNTDebug[3],
    CV4 => aCNTDebug[4],
    CV5 => aCNTDebug[5],
    CV6 => aCNTDebug[6],
    CV7 => aCNTDebug[7]); // FB_DEBUG_CounterArray
aCNTDebug[1] := fbDebugCNT.CV1;
END_ACTION

END_FUNCTION_BLOCK

// ---- POUs/METS/Common LIB/02_OUTER LIB/Outer FBs/FB_OUTER_ValidateOuterForReject.TcPOU
 (* scan for and validate Outers marked as requiring validation *)
FUNCTION_BLOCK FB_OUTER_ValidateOuterForReject
VAR_INPUT
	bExecute					: BOOL;			(* scan for completed Outer *)
	stCTDateTime				: ST_SYSTEM_DateTime;	(* CaseTrace date/time structure *)
	bValidateOCVOnly			: BOOL;
	bEnableRestoreOCV			: BOOL;
END_VAR
VAR_IN_OUT
	stProductInstruction		: ST_PCM_Status;					(* Product Instruction *)
	nSecquentionalCounter	: UDINT;
	stCodeInfo_Outer			: ST_CodeInfo;
	stOuterStatus				: ST_OUTER_Status;	(* Outer status *)
	stOuterStatusForRestore	: ST_OUTER_Status;	(* Outer status *)
	stOuterRejectReasons		: ST_RejectReasonsForOuter;
	stOuterStatusHMI			: ST_HMI_OuterStatus;
END_VAR
VAR_OUTPUT
	bDone						: BOOL;			(* TRUE = validation complete *)
	bBusy						: BOOL;			(* TRUE = validation in progress *)
	bError						: BOOL;			(* TRUE = validation error *)
	nErrorID					: UDINT;		(* error ID *)

	sRejectCode				: T_RejectCode;
	nRejectID					: UINT;
	bRejectOuter				: BOOL;
END_VAR
VAR
	fbExecute					: R_TRIG;
	(*sRetailSKU					: T_CodeRSKU;*)
	sLastBarcode				: T_OUTER_Barcode;
	nPackIndex				: INT;
	nCheckIndex				: INT;
	nDuplicatePairs			: INT;
	stSystemTime				: TIMESTRUCT;

	nTest			:INT;


	aPackStatusValue		: ARRAY[0..10] OF INT;
	aRejectCodePointer      : ARRAY[0..10] OF STRING(10);
	nRejectIndex			: INT;

	fbValidateOuter		: FB_CODE_ValidateExplicitCode;
	fbValidatePack			: FB_CODE_ValidateExplicitCode;

	bDuplicateFound		: BOOL;
	nGoodPackReads		: INT;
END_VAR

(* monitor rising edge of bExecute *)
fbExecute(CLK := bExecute);

(*stSystemTime := stCTDateTime.sSystemTime;*)

(* scan for completed Outers when validation is active *)
IF fbExecute.Q = TRUE THEN

	(* update outputs *)
	bDone := FALSE;
	bBusy := TRUE;
	bError := FALSE;
	nErrorID := 0;

	sRejectCode := '';
	bRejectOuter := FALSE;
	nRejectID	:= 0;

	(* validate OAC data *)
	stOuterStatus.stOACData.CodingAndTrackingMode := stProductInstruction.nOpMode;

	(* extract RetailSKU and SerialCode *)
	fbValidateOuter(	sFullCode := stOuterStatus.stOACData.Barcode,
						stCodeInfo := stCodeInfo_Outer,
						stProductInstruction := stProductInstruction);

	(*sRetailSKU	:= fbValidateOuter.sRsku;*)

	IF bValidateOCVOnly THEN

		nGoodPackReads	:=  stOuterStatus.stOACData.NumberOfLinkedPacks;

		IF  nGoodPackReads = stOuterStatus.stOACData.NumberOfPacks THEN

			FOR nPackIndex := 1 TO stOuterStatus.stOACData.NumberOfPacks DO

				IF stOuterStatus.aOACPackStatus[nPackIndex]  <> 2 	THEN

					(* Outer is valid, update status *)
					stOuterStatus.bOuterCodeValid := TRUE;
					stOuterStatus.bPackCodesValid := TRUE;

					sRejectCode := 'OK';
					nRejectID		:= 0;
				ELSE

					(* Outer is valid, update status *)
					stOuterStatus.bOuterCodeValid := FALSE;
					stOuterStatus.bPackCodesValid := FALSE;

					bError := TRUE;
					nErrorID := 20;
					sRejectCode 	:=	stOuterRejectReasons.stOuterPackCodeInvalid.sMetsDisplayCode;
					nRejectID		:= 	stOuterRejectReasons.stOuterPackCodeInvalid.nRejectID;

					EXIT;
				END_IF
			END_FOR
		ELSE
			(* update status *)
			bError := TRUE;
			nErrorID := 21;

			aPackStatusValue[0] := 	nGoodPackReads;
			aPackStatusValue[1] := 	stOuterStatus.stOACData.NumberOfPacks;
			aRejectCodePointer[0] := 'n1';
			aRejectCodePointer[1] := 'n2';

			sRejectCode 	:=	F_CODE_AssignValToString(stOuterRejectReasons.stOuterPackCodeNotRead.sMetsDisplayCode, aPackStatusValue, aRejectCodePointer);
			nRejectID		:= 	stOuterRejectReasons.stOuterPackCodeNotRead.nRejectID;
		END_IF

	ELSIF stOuterStatus.stOACData.OuterRejectCode <> 'OK' THEN

		bError := TRUE;
		nErrorID := 10;

		sRejectCode 	:= stOuterStatus.stOACData.OuterRejectCode;
		nRejectID		:= stOuterStatus.stOACData.OuterRejectID;
	ELSIF  stProductInstruction.nOpMode >= 7 AND sLastBarcode = stOuterStatus.stOACData.Barcode  AND stOuterStatus.stOACData.Barcode <> '' THEN

		bError := TRUE;
		nErrorID := 11;

		sRejectCode :=  stOuterRejectReasons.stOuterBarcodeDuplicate.sMetsDisplayCode;
		nRejectID		:= stOuterRejectReasons.stOuterBarcodeDuplicate.nRejectID;

	ELSIF stProductInstruction.nOpMode = 7
		AND fbValidateOuter.bValidationOK = TRUE THEN

		(* Outer is valid, update status *)
		stOuterStatus.bOuterCodeValid := TRUE;
		sRejectCode 	:= 'OK';
		nRejectID		:= 0;

	ELSIF stProductInstruction.nOpMode = 11
		AND fbValidateOuter.bValidationOK = TRUE THEN

		(* Outer is valid, update status *)
		stOuterStatus.bOuterCodeValid := TRUE;
		sRejectCode 	:= 'OK';
		nRejectID		:= 0;
		nGoodPackReads := 0;

		(*Restore missing data from OCV struct - do not reject outer*)
		IF bEnableRestoreOCV AND stOuterStatus.nStatus.16 = TRUE  AND stOuterStatusForRestore.nStatus.16 = FALSE THEN

			sRejectCode := 'OK - attempt to restore Pack (OCV) Data';
			stOuterStatus.bPackCodesValid := TRUE;
		(* <NumberOfPacks> > 0 *)
		ELSIF stOuterStatus.stOACData.NumberOfLinkedPacks > 0 THEN
			(*nGoodPackReads := 0;*)
			(* <nGoodPackReads>  > <AcceptanceLevel> *)
			FOR nPackIndex := 1 TO stOuterStatus.stOACData.NumberOfPacks DO

(*alternativly we could check********************************************************************************
		IF NOT stOuterStatus.stOACData.PackCodeStatus[nPackIndex].1 		AND
			NOT stOuterStatus.stOACData.PackCodeStatus[nPackIndex].2	AND
			NOT stOuterStatus.stOACData.PackCodeStatus[nPackIndex].3	THEN

					IF stOuterStatus.stOACData.PackCodeStatus[nPackIndex].5 		OR 
						stOuterStatus.stOACData.PackCodeStatus[nPackIndex].6 		OR 
						stOuterStatus.stOACData.PackCodeStatus[nPackIndex].9 		OR 
						stOuterStatus.stOACData.PackCodeStatus[nPackIndex].10	THEN
***************************************************************************************************************)

				IF stOuterStatus.aOACPackStatus[nPackIndex]  <> 1 		AND
					stOuterStatus.aOACPackStatus[nPackIndex]  <> 2 	AND
					stOuterStatus.aOACPackStatus[nPackIndex]  <> 3 	THEN

					IF stOuterStatus.aOACPackStatus[nPackIndex]  > 4  	THEN
						nGoodPackReads := nGoodPackReads + 1;
					END_IF
				ELSE
					nGoodPackReads := -1;
					EXIT;
				END_IF
			END_FOR

		(* sufficient number of Pack codes read and valid, update status *)
			IF nGoodPackReads >= stOuterStatus.stOACData.AcceptanceLevel THEN
				stOuterStatus.bPackCodesValid := TRUE;

				FOR nPackIndex := 1 TO stOuterStatus.stOACData.NumberOfPacks DO

					IF  stOuterStatus.aOACPackStatus[nPackIndex]  = 0 THEN

							stOuterStatus.stOACData.PackCode[nPackIndex] 			:= F_CODE_BATSerializator(stCTDateTime, ePack, TRUE, stProductInstruction, nSecquentionalCounter);
							(* change status to indicate no read in an accepted outer *)
							stOuterStatus.aOACPackStatus[nPackIndex]				:= 5 (*4 - for now avoid 4 as PackStatus is check in several places and has to be 5*);
							(*additional bit passing to CAC*)
							stOuterStatus.stOACData.PackCodeStatus[nPackIndex]:=
														F_FiltredSetBitState16(TRUE, 'LOW', 4, TRUE, stOuterStatus.stOACData.PackCodeStatus[nPackIndex]);

							stOuterStatus.stOACData.PackRejectCode[nPackIndex]   	:= 'OK';
							stOuterStatus.stOACData.PackRejectID[nPackIndex]		:= 0;
					END_IF
				END_FOR
				(*NumberOfLinkedPacks we modify only in final case content validation*)

		(* invalid pack code(s) found *)
			ELSIF nGoodPackReads = -1 THEN
								(* update status *)
				bError := TRUE;
				nErrorID := 22;
				sRejectCode 	:=	stOuterRejectReasons.stOuterPackCodeInvalid.sMetsDisplayCode;
				nRejectID		:= 	stOuterRejectReasons.stOuterPackCodeInvalid.nRejectID;
		(* insufficient pack codes read *)
			ELSE
				(* update status *)
				bError := TRUE;
				nErrorID := 23;

				aPackStatusValue[0] := 	nGoodPackReads;
				aPackStatusValue[1] := 	stOuterStatus.stOACData.NumberOfPacks;
				aRejectCodePointer[0] := 'n1';
				aRejectCodePointer[1] := 'n2';

				sRejectCode 	:=	F_CODE_AssignValToString(stOuterRejectReasons.stOuterPackCodeNotRead.sMetsDisplayCode, aPackStatusValue, aRejectCodePointer);
				nRejectID		:= 	stOuterRejectReasons.stOuterPackCodeNotRead.nRejectID;
			END_IF
		(* <NumberOfPacks> invalid *)
		ELSE
			(* update status *)
			bError := TRUE;
			nErrorID := 24;
			sRejectCode	 := 	stOuterRejectReasons.stOuterPackCodeDataNotFound.sMetsDisplayCode;
			nRejectID		:= 	stOuterRejectReasons.stOuterPackCodeDataNotFound.nRejectID;
		END_IF
	(* code is invalid *)
	ELSIF stOuterStatus.stOACData.Barcode <> '' THEN
		(* update outputs *)
		bError := TRUE;
		nErrorID := 12;
		IF fbValidateOuter.bGtinOK = FALSE THEN
			sRejectCode := stOuterRejectReasons.stOuterBarcodeGtinError.sMetsDisplayCode;
			nRejectID		:= 	stOuterRejectReasons.stOuterBarcodeGtinError.nRejectID;
		ELSIF fbValidateOuter.bBrandOK = FALSE THEN
			sRejectCode := stOuterRejectReasons.stOuterCodesBrandSpecError.sMetsDisplayCode;
			nRejectID		:= 	stOuterRejectReasons.stOuterCodesBrandSpecError.nRejectID;
		ELSIF fbValidateOuter.bRskuOK = FALSE THEN
			sRejectCode := stOuterRejectReasons.stOuterBarcodeRskuError.sMetsDisplayCode;
			nRejectID		:= 	stOuterRejectReasons.stOuterBarcodeRskuError.nRejectID;
		ELSIF fbValidateOuter.bSerialCodeOK = FALSE THEN
			sRejectCode := stOuterRejectReasons.stOuterCodeSerialError.sMetsDisplayCode;
			nRejectID		:= 	stOuterRejectReasons.stOuterCodeSerialError.nRejectID;
		ELSE
			sRejectCode :=  stOuterRejectReasons.stOuterBarcodeInvalidLength.sMetsDisplayCode;
			nRejectID		:= 	stOuterRejectReasons.stOuterBarcodeInvalidLength.nRejectID;
		END_IF

	(* no code read *)
	ELSE
		(* update outputs *)
		bError := TRUE;
		nErrorID := 13;
		sRejectCode := stOuterRejectReasons.stOuterBarcodeNotRead.sMetsDisplayCode;
		nRejectID		:= 	stOuterRejectReasons.stOuterBarcodeNotRead.nRejectID;

	END_IF


(**************** update Outer status *******************)
	stOuterStatus.nStatus.10 := FALSE;
	stOuterStatus.nStatus.11 := FALSE;

	IF stOuterStatus.bQAReject THEN
		sRejectCode 	:= stOuterRejectReasons.stOuterQAReject.sMetsDisplayCode;
		nRejectID		:= 	stOuterRejectReasons.stOuterQAReject.nRejectID;
	END_IF

	(* CaseTrace mode, Outer code must be valid *)
	IF stProductInstruction.nOpMode = 7 AND stOuterStatus.bOuterCodeValid = TRUE AND stOuterStatus.bQAReject = FALSE THEN
		(* Outer is valid *)
		stOuterStatus.nStatus.10 := TRUE;
		bRejectOuter := FALSE;

	(* PackTrace mode, Outer code and Pack codes must be valid *)
	ELSIF stProductInstruction.nOpMode  = 11 AND stOuterStatus.bOuterCodeValid = TRUE AND stOuterStatus.bPackCodesValid = TRUE AND stOuterStatus.bQAReject = FALSE THEN
		(* Outer is valid *)
		stOuterStatus.nStatus.10 := TRUE;
		bRejectOuter := FALSE;

	(* Outer has failed validation *)
	ELSE

		(* Outer is invalid *)
		stOuterStatus.nStatus.11 := TRUE;
		bRejectOuter := TRUE;
	END_IF

	stOuterStatus.stOACData.OuterRejectCode := sRejectCode;
	stOuterStatus.stOACData.OuterRejectID	:= nRejectID;

	stOuterStatusHMI.sBarcode := stOuterStatus.stOACData.Barcode;

	stOuterStatusHMI.sProductionDate := 	stOuterStatus.stOACData.ProductionDate;
	stOuterStatusHMI.sProductionTime :=		stOuterStatus.stOACData.ProductionTime;

	MEMMOVE(ADR(stOuterStatusHMI.aPackCode), ADR(stOuterStatus.stOACData.PackCode), SIZEOF(stOuterStatus.stOACData.PackCode));
	MEMMOVE(ADR(stOuterStatusHMI.aOACPackStatus), ADR(stOuterStatus.aOACPackStatus), SIZEOF(stOuterStatus.aOACPackStatus));

(* 7 for now see asigmnet on screen - after leave 5*)
	FOR nPackIndex := 1 TO stOuterStatus.stOACData.NumberOfPacks DO

		IF  stOuterStatus.stOACData.PackCodeStatus[nPackIndex].4 THEN
			stOuterStatusHMI.aOACPackStatus[nPackIndex]	:= 7;
		END_IF
	END_FOR

	MEMMOVE(ADR(stOuterStatusHMI.aPackRejectCode), ADR(stOuterStatus.stOACData.PackRejectCode), SIZEOF(stOuterStatus.stOACData.PackRejectCode));
	MEMMOVE(ADR(stOuterStatusHMI.aPackRejectID), ADR(stOuterStatus.stOACData.PackRejectID), SIZEOF(stOuterStatus.stOACData.PackRejectID));

	stOuterStatusHMI.nNumberOfPacks			:=	stOuterStatus.stOACData.NumberOfPacks;
	stOuterStatusHMI.nAcceptanceLevel			:=	stOuterStatus.stOACData.AcceptanceLevel;
	stOuterStatusHMI.nNumberOfLinkedPacks	:=	SEL(nGoodPackReads = -1, nGoodPackReads, 0) ;

	stOuterStatusHMI.sOuterRejectCode	:= stOuterStatus.stOACData.OuterRejectCode;
	stOuterStatusHMI.nOuterRejectID		:= stOuterStatus.stOACData.OuterRejectID;

	sLastBarcode := stOuterStatus.stOACData.Barcode;

	(* update outputs *)
	bDone := TRUE;
	bBusy := FALSE;

(* no action required *)
ELSIF bExecute = FALSE THEN

	(* reset outputs *)
	bDone := FALSE;
	bBusy := FALSE;
	bError := FALSE;
	(*nErrorID := 0;*)
	bRejectOuter := FALSE;
END_IF

END_FUNCTION_BLOCK

// ---- POUs/METS/Common LIB/08_SOFTWARE LIB/AI Codes And Validation FBs/F_CODE_AssignValToString.TcPOU
FUNCTION F_CODE_AssignValToString : T_MaxString
VAR_INPUT
	asRejectReason		: T_MaxString;
	anValue				: ARRAY[0..10] OF INT;
	asPointer          	  		: ARRAY[0..10] OF STRING(10);
END_VAR

VAR
	(*bPointerNotFound	           : BOOL;*)
	nCounter				: INT;
	nPointerPos			: INT;
	asAssignedRejectReason	: T_MaxString;
END_VAR

(* This Function assigns value to predefined Pointer in string.
     Function can assing up to 10 Values
     For ex. string Reject Reason := 'XXDUPn1-n2XX'
     	         nValue := [3, 4], sPointer := ['n1', 'n2']		
	         asRejectReason := 'XXDUP3-4XX'	*)

F_CODE_AssignValToString := '';

asAssignedRejectReason := asRejectReason;

REPEAT
	nPointerPos := FIND(asAssignedRejectReason, asPointer[nCounter]);
	IF nPointerPos > 0 AND  asPointer[nCounter] <> '' THEN
		 asAssignedRejectReason := REPLACE(asAssignedRejectReason, INT_TO_STRING(anValue[nCounter]) , LEN(asPointer[nCounter]), nPointerPos);
	END_IF;
	nCounter := nCounter + 1;
UNTIL
	nCounter >= 10
END_REPEAT

IF nCounter <> 0 THEN
	F_CODE_AssignValToString := asAssignedRejectReason;
ELSE
	F_CODE_AssignValToString := asRejectReason;
END_IF;

END_FUNCTION

